_CFC_ (* Continuous Function Chart, elements in execution order *)
(* VÄRMEREGLERING *)
(* PUMPSTYRNING *)
(* BÖRVÄRDESKURVA *)
(* LARM/AVVIKELSELARM *)
#0 HUS1_VS20_SO(bManover: HUS2_AS01_SOMMARVINTER.bVINTER_TILL)
#1 HUS1_VS20_PV01(_bAuto: #0.bTILL)
#2 HUS1_VS20_PV01_M <= #1._bMANOVER
#3 HUS1_VS20_PV01_LD <= #1._bDRIFTFEL
#4 HUS1_VS20_PV01_LM <= #1._bLHAND
#5 SUB(HUS1_VS20_GT11_BB, HUS1_VS20_GT11_BB1)
#6 HUS1_VS20_GT11_PID(_bEnable: #0.bTILL, _rBV: #5, _rMV: HUS1_VS20_GT11_MV)
#7 HUS1_VS20_SV21_R <= #6._rY1
#8 HUS1_VS20_GT11_KURVA(_rGT3N: HUS2_AS01_GT31_MV)
#9 HUS1_VS20_GT11_BB <= #8._rBB
#10 HUS1_VS20_EFFEKTBEGR(_rGT3N: HUS2_AS01_GT31_MV, _rMQ41_SV: HUS2_VP1.SV_MQ41)
#11 HUS1_VS20_GT11_BB1 <= #10._rBB
#12 HUS1_VS20_GT11_larm()
_END_CFC_
(* the same logic as Structured Text *)
(* VÄRMEREGLERING *)
(* PUMPSTYRNING *)
(* BÖRVÄRDESKURVA *)
(* LARM/AVVIKELSELARM *)
HUS1_VS20_SO(bManover := HUS2_AS01_SOMMARVINTER.bVINTER_TILL);
HUS1_VS20_PV01(_bAuto := HUS1_VS20_SO.bTILL);
HUS1_VS20_PV01_M := HUS1_VS20_PV01._bMANOVER;
HUS1_VS20_PV01_LD := HUS1_VS20_PV01._bDRIFTFEL;
HUS1_VS20_PV01_LM := HUS1_VS20_PV01._bLHAND;
HUS1_VS20_GT11_PID(_bEnable := HUS1_VS20_SO.bTILL, _rBV := HUS1_VS20_GT11_BB - HUS1_VS20_GT11_BB1, _rMV := HUS1_VS20_GT11_MV);
HUS1_VS20_SV21_R := HUS1_VS20_GT11_PID._rY1;
HUS1_VS20_GT11_KURVA(_rGT3N := HUS2_AS01_GT31_MV);
HUS1_VS20_GT11_BB := HUS1_VS20_GT11_KURVA._rBB;
HUS1_VS20_EFFEKTBEGR(_rGT3N := HUS2_AS01_GT31_MV, _rMQ41_SV := HUS2_VP1.SV_MQ41);
HUS1_VS20_GT11_BB1 := HUS1_VS20_EFFEKTBEGR._rBB;
HUS1_VS20_GT11_larm();
END_PROGRAM

(* POU SYSTEM/VS20/HUS1_VS20_SO, CFC *)
PROGRAM HUS1_VS20_SO
VAR_INPUT

	bManover: BOOL;
END_VAR

VAR
	SERVICEOMKOPPLARE: fbManualOverride;

	UPPSTARTSSEKVENSIERING: BOOL;
END_VAR

VAR_OUTPUT
	bTILL:BOOL;

END_VAR
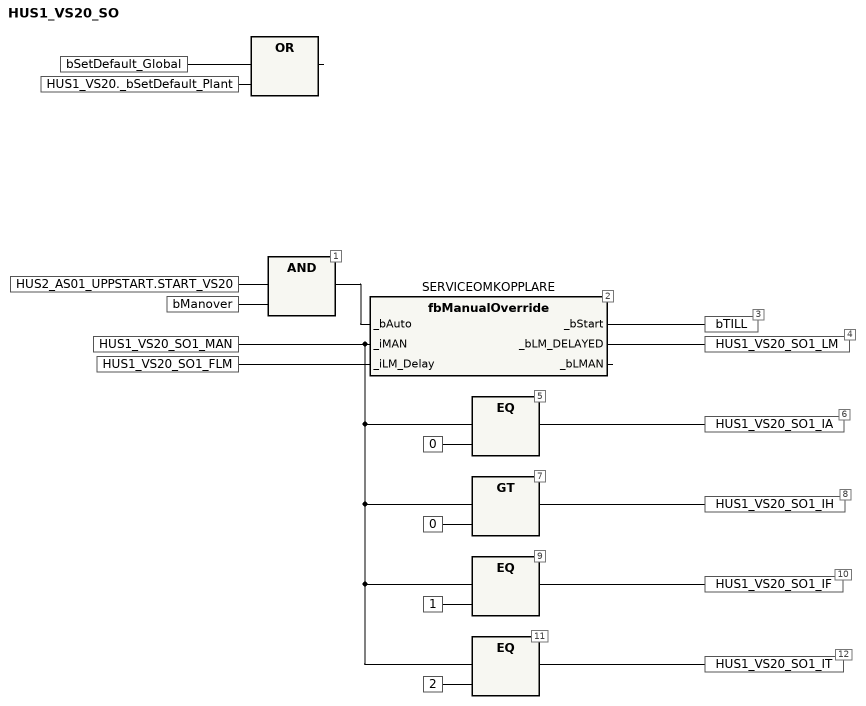
_CFC_ (* Continuous Function Chart, elements in execution order *)
#0 OR(bSetDefault_Global, HUS1_VS20._bSetDefault_Plant)
#1 AND(HUS2_AS01_UPPSTART.START_VS20, bManover)
#2 SERVICEOMKOPPLARE:fbManualOverride(_bAuto: #1, _iMAN: HUS1_VS20_SO1_MAN, _iLM_Delay: HUS1_VS20_SO1_FLM)
#3 bTILL <= #2._bStart
#4 HUS1_VS20_SO1_LM <= #2._bLM_DELAYED
#5 EQ(HUS1_VS20_SO1_MAN, 0)
#6 HUS1_VS20_SO1_IA <= #5
#7 GT(HUS1_VS20_SO1_MAN, 0)
#8 HUS1_VS20_SO1_IH <= #7
#9 EQ(HUS1_VS20_SO1_MAN, 1)
#10 HUS1_VS20_SO1_IF <= #9
#11 EQ(HUS1_VS20_SO1_MAN, 2)
#12 HUS1_VS20_SO1_IT <= #11
_END_CFC_
(* the same logic as Structured Text *)
(* result unused: bSetDefault_Global OR HUS1_VS20._bSetDefault_Plant *)
SERVICEOMKOPPLARE(_bAuto := HUS2_AS01_UPPSTART.START_VS20 AND bManover, _iMAN := HUS1_VS20_SO1_MAN, _iLM_Delay := HUS1_VS20_SO1_FLM);
bTILL := SERVICEOMKOPPLARE._bStart;
HUS1_VS20_SO1_LM := SERVICEOMKOPPLARE._bLM_DELAYED;
HUS1_VS20_SO1_IA := HUS1_VS20_SO1_MAN = 0;
HUS1_VS20_SO1_IH := HUS1_VS20_SO1_MAN > 0;
HUS1_VS20_SO1_IF := HUS1_VS20_SO1_MAN = 1;
HUS1_VS20_SO1_IT := HUS1_VS20_SO1_MAN = 2;
END_PROGRAM

(* POU SYSTEM/VS20/Pumpstyrning/HUS1_VS20_PV01, CFC *)
PROGRAM HUS1_VS20_PV01

VAR

	Default: BOOL;
	Motor: FB_HVACMotor1Speed;


	fbReset1: fbBool_Reset;
	AlarmDelay: fbDelayedAlarmSeconds;

	MANHAND: fbManualOverride;
END_VAR
VAR


(********************MOTOR********************)
(*INPUT*)
	eCtrlModeActuator			:E_HVACActuatorMode;
	tStartDelay						:TIME;
	tStopDelay						:TIME;
	tDelayFeedbContactor			:TIME:=T#30s;
	tFeedbProcessTimer				:TIME:=T#30s;
	tDelayFeedbProcess				:TIME:=T#30s;
(*OUTPUT*)
	byState							:BYTE ;
	bStateAuto							:BOOL;
	bStateRepairSwitch				:BOOL;
	bStateManSwitch				:BOOL;
	eStateModeActuator				:E_HVACActuatorMode;
	byError							:BYTE ;
	bErrorMotorprotec				:BOOL;
	bErrorFeedbContactor			:BOOL;
	bErrorFeedbProcess			:BOOL;
	bInvalidParameter				:BOOL;

END_VAR

VAR_INPUT
	_bAuto							:BOOL;(* enable function block *)
END_VAR

VAR_OUTPUT
	_bMANOVER						:BOOL;
	_bDRIFTFEL						:BOOL;
	_bLHAND							:BOOL;
END_VAR
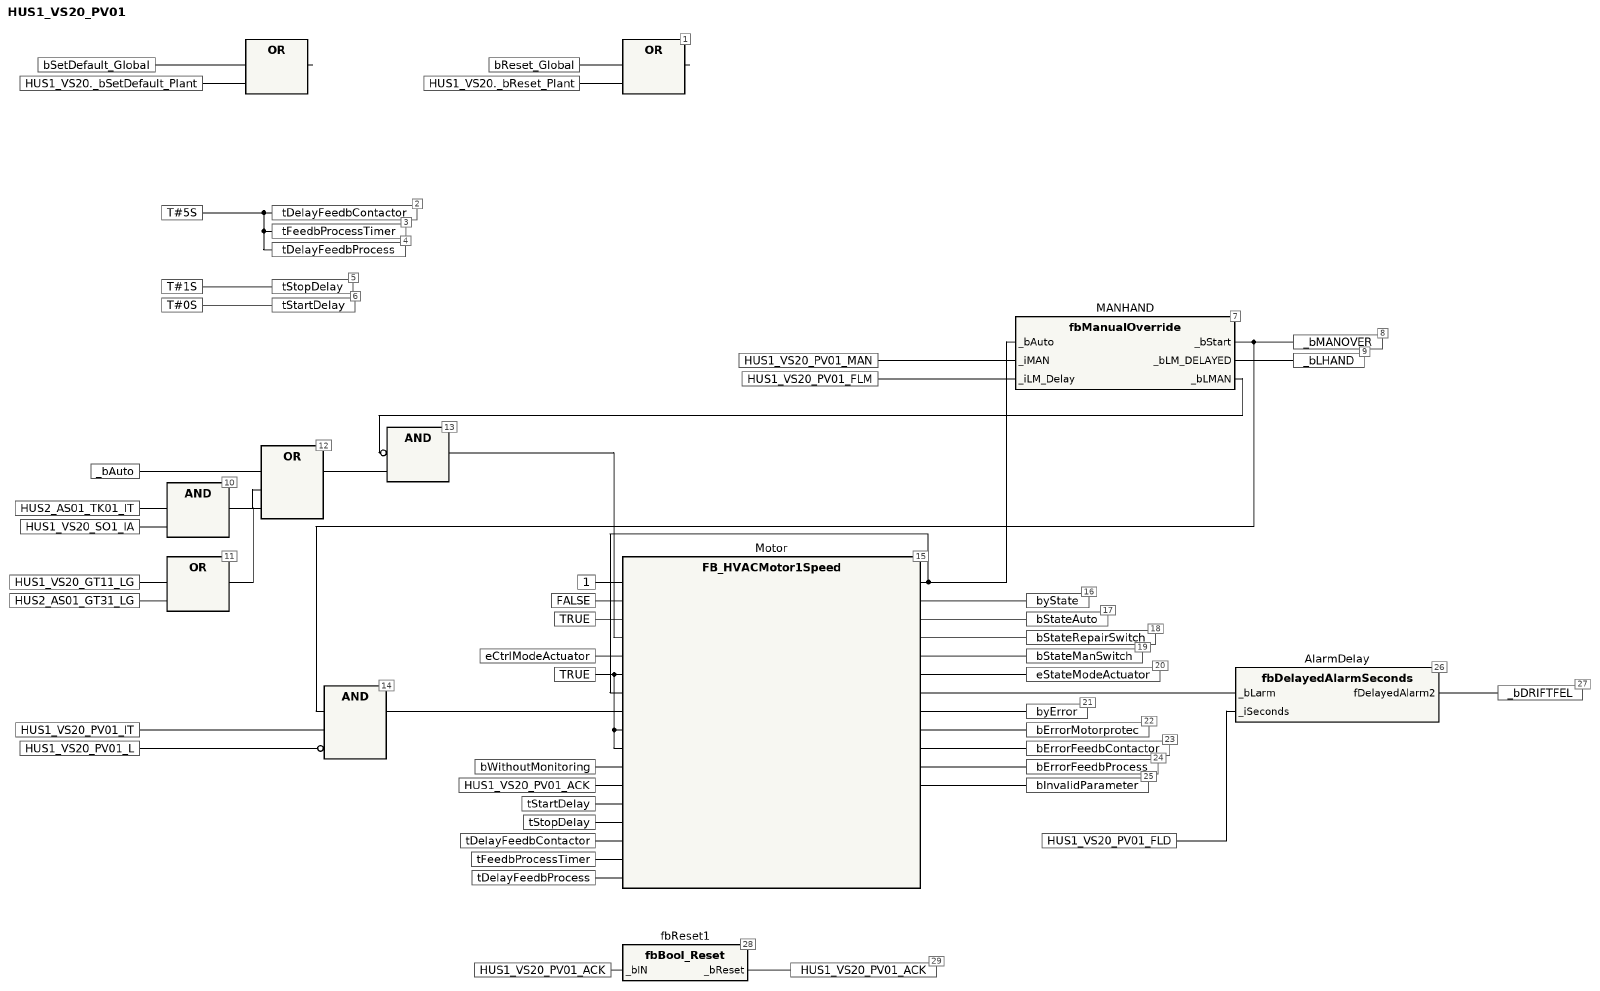
_CFC_ (* Continuous Function Chart, elements in execution order *)
#0 OR(bSetDefault_Global, HUS1_VS20._bSetDefault_Plant)
#1 OR(bReset_Global, HUS1_VS20._bReset_Plant)
#2 tDelayFeedbContactor <= T#5S
#3 tFeedbProcessTimer <= T#5S
#4 tDelayFeedbProcess <= T#5S
#5 tStopDelay <= T#1S
#6 tStartDelay <= T#0S
#7 MANHAND:fbManualOverride(_bAuto: #15.out 1, _iMAN: HUS1_VS20_PV01_MAN, _iLM_Delay: HUS1_VS20_PV01_FLM)
#8 _bMANOVER <= #7._bStart
#9 _bLHAND <= #7._bLM_DELAYED
#10 AND(HUS2_AS01_TK01_IT, HUS1_VS20_SO1_IA)
#11 OR(HUS1_VS20_GT11_LG, HUS2_AS01_GT31_LG)
#12 OR(_bAuto, #10, #11)
#13 AND(NOT #7._bLMAN, #12)
#14 AND(#7._bStart, HUS1_VS20_PV01_IT, NOT HUS1_VS20_PV01_L)
#15 Motor:FB_HVACMotor1Speed(1, FALSE, TRUE, #13, eCtrlModeActuator, TRUE, #15.out 1, #14, TRUE, TRUE, bWithoutMonitoring, HUS1_VS20_PV01_ACK, tStartDelay, tStopDelay, tDelayFeedbContactor, tFeedbProcessTimer, tDelayFeedbProcess)
#16 byState <= #15.out 2
#17 bStateAuto <= #15.out 3
#18 bStateRepairSwitch <= #15.out 4
#19 bStateManSwitch <= #15.out 5
#20 eStateModeActuator <= #15.out 6
#21 byError <= #15.out 8
#22 bErrorMotorprotec <= #15.out 9
#23 bErrorFeedbContactor <= #15.out 10
#24 bErrorFeedbProcess <= #15.out 11
#25 bInvalidParameter <= #15.out 12
#26 AlarmDelay:fbDelayedAlarmSeconds(_bLarm: #15.out 7, _iSeconds: HUS1_VS20_PV01_FLD)
#27 _bDRIFTFEL <= #26.fDelayedAlarm2
#28 fbReset1:fbBool_Reset(_bIN: HUS1_VS20_PV01_ACK)
#29 HUS1_VS20_PV01_ACK <= #28._bReset
_END_CFC_
END_PROGRAM

(* POU SYSTEM/VS20/Tempreglering/HUS1_VS20_GT11_PID, FAI *)
PROGRAM HUS1_VS20_GT11_PID

VAR_INPUT
	_bEnable		:BOOL;
	_rBV			:REAL;
	_rMV			:REAL;
END_VAR

VAR_OUTPUT
	_rY1                         : REAL;
END_VAR


VAR
	_bSetDefaultPID:BOOL;
	_bReset_Local:BOOL;


	SVX: FB_HVACPIDCtrl;
	eDataSecurityType         : E_HVACDataSecurityType;
	rInitialValue            : REAL;
	bResetController          : BOOL;
	_eCtrlMode				:E_HVACCtrlMode;(*
									eHVACCtrlMode_Auto      := 0,
								   	eHVACCtrlMode_Manual   := 1 *)
	_rOverrideValue			:REAL;(* controller output rY in operating mode eCtrlMode =1 *)
	rXW                        : REAL;
	bMaxLimit                  : BOOL;
	bMinLimit                  : BOOL;
	bActive                    : BOOL;
	bARWactive                 : BOOL;
	eState                     : E_HVACState;
	bError                     : BOOL;
	eErrorCode                 : E_HVACErrorCodes;
	bInvalidParameter          : BOOL;

	bDirection              : BOOL;
	_rKP: REAL;
	_rCH: REAL;
	tTi                     : TIME;
	tTv                     : TIME;
	tTd                     : TIME;

	rYMin                   : REAL;
	rYMax                   : REAL;

	CI: fbBer_PID_inst;
	CS: fbBer_PID_inst;
	CD: fbBer_PID_inst;

	fbPersistent_CH: FB_HVACPersistent_Real;
	fbPersistent_CP: FB_HVACPersistent_Real;
	fbPersistent_CI: FB_HVACPersistent_Real;
	fbPersistent_CS: FB_HVACPersistent_Real;
	fbPersistent_CD: FB_HVACPersistent_Real;
	LM_DELAY: fbDelayedAlarmMinutes;
END_VAR
(* body not read: cfc97 *)
END_PROGRAM

(* POU SYSTEM/VS20/Börvärden & kurvor/HUS1_VS20_GT11_KURVA, FAI *)
PROGRAM HUS1_VS20_GT11_KURVA
VAR
(****************************************** heating curve **********************************************************************************************************************)

	_bSetDefaultHC			:BOOL;


	fbScale_n:			FB_HVACScale_nPoint;
	_bErrParam:			BOOL;								(*ParameterError*)
	stScaleParameter:	ST_HVACParameterScale_nPoint	;	(*Parameter struktur på antal brutpunkter*)


	fbTemp1:	FB_HVACPersistent_Real;
	fbTemp2:	FB_HVACPersistent_Real;
	fbTemp3:	FB_HVACPersistent_Real;
	fbTemp4:	FB_HVACPersistent_Real;
	fbTemp5:	FB_HVACPersistent_Real;

	fbOutsideTemp1:	FB_HVACPersistent_Real;
	fbOutsideTemp2:	FB_HVACPersistent_Real;
	fbOutsideTemp3:	FB_HVACPersistent_Real;
	fbOutsideTemp4:	FB_HVACPersistent_Real;
	fbOutsideTemp5:	FB_HVACPersistent_Real;
	BB_min: FB_HVACPersistent_Real;
	BB_max: FB_HVACPersistent_Real;

END_VAR

VAR_INPUT
	_rGT3N	:REAL; (*Utegivare*)

END_VAR

VAR_OUTPUT
	_rBB		:LREAL;
END_VAR
(* body not read: cfc97 *)
END_PROGRAM

(* POU SYSTEM/VS20/Börvärden & kurvor/HUS1_VS20_EFFEKTBEGR, FAI *)
PROGRAM HUS1_VS20_EFFEKTBEGR
VAR
(****************************************** heating curve **********************************************************************************************************************)

	_bSetDefaultHC			:BOOL;


	fbScale_n:			FB_HVACScale_nPoint;
	_bErrParam:			BOOL;								(*ParameterError*)
	stScaleParameter:	ST_HVACParameterScale_nPoint	;	(*Parameter struktur på antal brutpunkter*)


	fbTemp1:	FB_HVACPersistent_Real;
	fbTemp2:	FB_HVACPersistent_Real;
	fbTemp3:	FB_HVACPersistent_Real;
	fbTemp4:	FB_HVACPersistent_Real;
	fbTemp5:	FB_HVACPersistent_Real;

	fbOutsideTemp1:	FB_HVACPersistent_Real;
	fbOutsideTemp2:	FB_HVACPersistent_Real;
	fbOutsideTemp3:	FB_HVACPersistent_Real;
	fbOutsideTemp4:	FB_HVACPersistent_Real;
	fbOutsideTemp5:	FB_HVACPersistent_Real;
	BB_min: FB_HVACPersistent_Real;
	BB_max: FB_HVACPersistent_Real;

	CalcForskjutning: fbConversionScale;
	MIN_LIMIT: REAL;
END_VAR

VAR_INPUT
	_rGT3N	:REAL; (*Utegivare*)
	_rMQ41_SV	:REAL;

END_VAR

VAR_OUTPUT
	_rBB		:LREAL;
END_VAR
(* body not read: cfc97 *)
END_PROGRAM

(* POU SYSTEM/VS20/Larm/HUS1_VS20_GT11_LARM, FAI *)
PROGRAM HUS1_VS20_GT11_LARM

VAR_OUTPUT
	_bLSumma					: BOOL;	(*Summalarm*)

END_VAR
VAR

	_bSetDefault: 				BOOL;		(*Se default values*)
	fbLarm: fbAvvikelselarm;


	fbHigh: FB_HVACPersistent_Real;
	fbAlarmDelayLH: FB_HVACPersistent_Int;
	fbLow: FB_HVACPersistent_Real;
	fbAlarmDelayLL: FB_HVACPersistent_Int;


END_VAR
(* body not read: cfc97 *)
END_PROGRAM

(* POU SYSTEM/VS30/HUS2_VS30, CFC *)
PROGRAM HUS2_VS30
VAR
	_bSetDefault_Plant		:BOOL;
	_bReset_Plant				:BOOL;

END_VAR
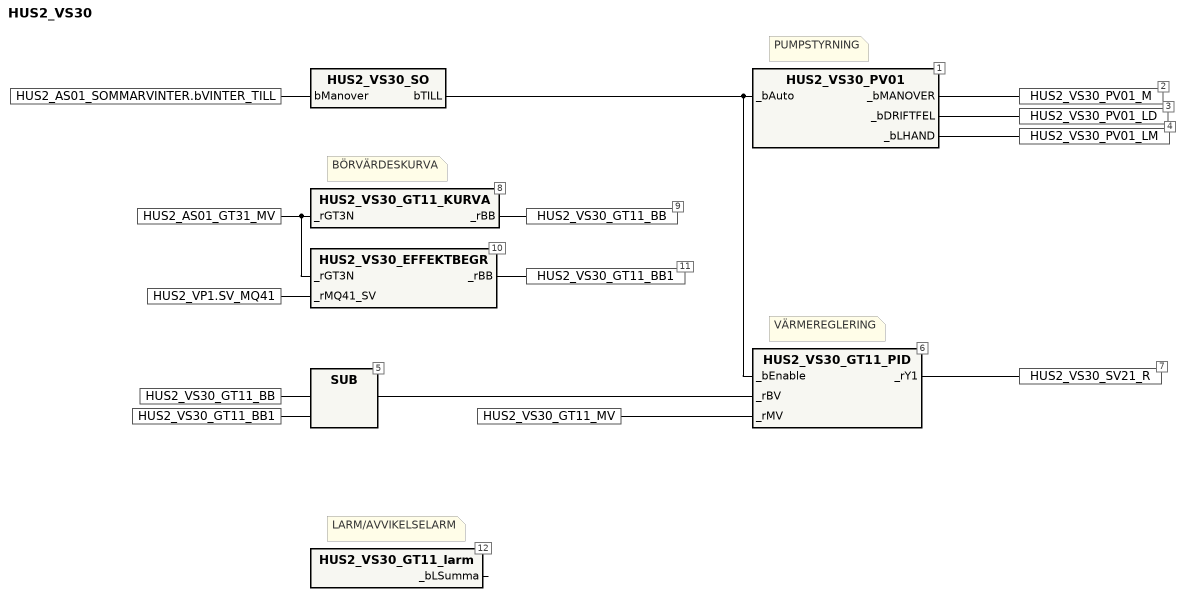
_CFC_ (* Continuous Function Chart, elements in execution order *)
(* LARM/AVVIKELSELARM *)
(* BÖRVÄRDESKURVA *)
(* PUMPSTYRNING *)
(* VÄRMEREGLERING *)
#0 HUS2_VS30_SO(bManover: HUS2_AS01_SOMMARVINTER.bVINTER_TILL)
#1 HUS2_VS30_PV01(_bAuto: #0.bTILL)
#2 HUS2_VS30_PV01_M <= #1._bMANOVER
#3 HUS2_VS30_PV01_LD <= #1._bDRIFTFEL
#4 HUS2_VS30_PV01_LM <= #1._bLHAND
#5 SUB(HUS2_VS30_GT11_BB, HUS2_VS30_GT11_BB1)
#6 HUS2_VS30_GT11_PID(_bEnable: #0.bTILL, _rBV: #5, _rMV: HUS2_VS30_GT11_MV)
#7 HUS2_VS30_SV21_R <= #6._rY1
#8 HUS2_VS30_GT11_KURVA(_rGT3N: HUS2_AS01_GT31_MV)
#9 HUS2_VS30_GT11_BB <= #8._rBB
#10 HUS2_VS30_EFFEKTBEGR(_rGT3N: HUS2_AS01_GT31_MV, _rMQ41_SV: HUS2_VP1.SV_MQ41)
#11 HUS2_VS30_GT11_BB1 <= #10._rBB
#12 HUS2_VS30_GT11_larm()
_END_CFC_
(* the same logic as Structured Text *)
(* LARM/AVVIKELSELARM *)
(* BÖRVÄRDESKURVA *)
(* PUMPSTYRNING *)
(* VÄRMEREGLERING *)
HUS2_VS30_SO(bManover := HUS2_AS01_SOMMARVINTER.bVINTER_TILL);
HUS2_VS30_PV01(_bAuto := HUS2_VS30_SO.bTILL);
HUS2_VS30_PV01_M := HUS2_VS30_PV01._bMANOVER;
HUS2_VS30_PV01_LD := HUS2_VS30_PV01._bDRIFTFEL;
HUS2_VS30_PV01_LM := HUS2_VS30_PV01._bLHAND;
HUS2_VS30_GT11_PID(_bEnable := HUS2_VS30_SO.bTILL, _rBV := HUS2_VS30_GT11_BB - HUS2_VS30_GT11_BB1, _rMV := HUS2_VS30_GT11_MV);
HUS2_VS30_SV21_R := HUS2_VS30_GT11_PID._rY1;
HUS2_VS30_GT11_KURVA(_rGT3N := HUS2_AS01_GT31_MV);
HUS2_VS30_GT11_BB := HUS2_VS30_GT11_KURVA._rBB;
HUS2_VS30_EFFEKTBEGR(_rGT3N := HUS2_AS01_GT31_MV, _rMQ41_SV := HUS2_VP1.SV_MQ41);
HUS2_VS30_GT11_BB1 := HUS2_VS30_EFFEKTBEGR._rBB;
HUS2_VS30_GT11_larm();
END_PROGRAM

(* POU SYSTEM/VS30/HUS2_VS30_SO, CFC *)
PROGRAM HUS2_VS30_SO
VAR_INPUT

	bManover: BOOL;
END_VAR

VAR
	SERVICEOMKOPPLARE: fbManualOverride;

	UPPSTARTSSEKVENSIERING: BOOL;
END_VAR

VAR_OUTPUT
	bTILL:BOOL;

END_VAR
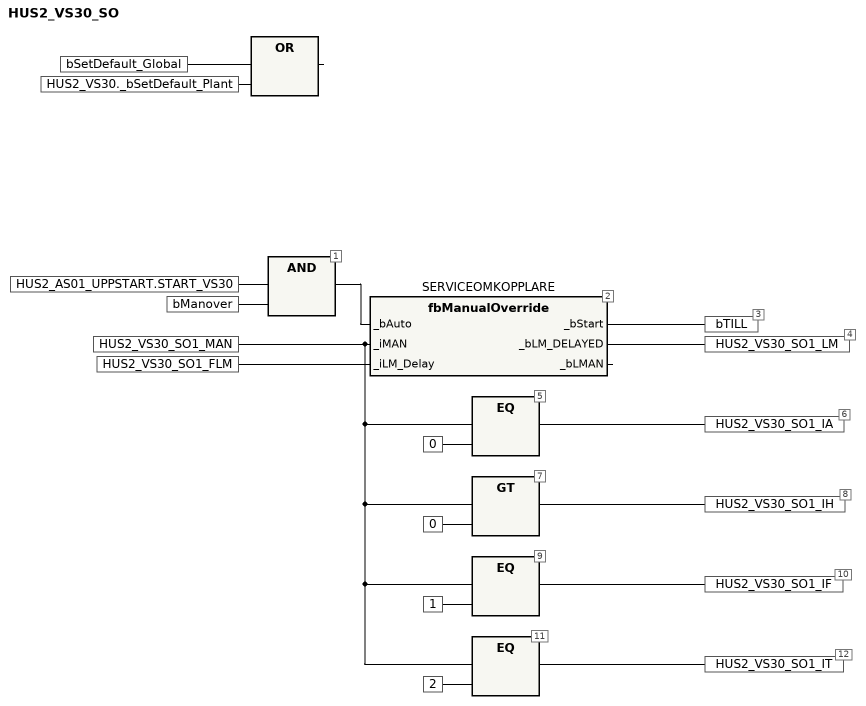
_CFC_ (* Continuous Function Chart, elements in execution order *)
#0 OR(bSetDefault_Global, HUS2_VS30._bSetDefault_Plant)
#1 AND(HUS2_AS01_UPPSTART.START_VS30, bManover)
#2 SERVICEOMKOPPLARE:fbManualOverride(_bAuto: #1, _iMAN: HUS2_VS30_SO1_MAN, _iLM_Delay: HUS2_VS30_SO1_FLM)
#3 bTILL <= #2._bStart
#4 HUS2_VS30_SO1_LM <= #2._bLM_DELAYED
#5 EQ(HUS2_VS30_SO1_MAN, 0)
#6 HUS2_VS30_SO1_IA <= #5
#7 GT(HUS2_VS30_SO1_MAN, 0)
#8 HUS2_VS30_SO1_IH <= #7
#9 EQ(HUS2_VS30_SO1_MAN, 1)
#10 HUS2_VS30_SO1_IF <= #9
#11 EQ(HUS2_VS30_SO1_MAN, 2)
#12 HUS2_VS30_SO1_IT <= #11
_END_CFC_
(* the same logic as Structured Text *)
(* result unused: bSetDefault_Global OR HUS2_VS30._bSetDefault_Plant *)
SERVICEOMKOPPLARE(_bAuto := HUS2_AS01_UPPSTART.START_VS30 AND bManover, _iMAN := HUS2_VS30_SO1_MAN, _iLM_Delay := HUS2_VS30_SO1_FLM);
bTILL := SERVICEOMKOPPLARE._bStart;
HUS2_VS30_SO1_LM := SERVICEOMKOPPLARE._bLM_DELAYED;
HUS2_VS30_SO1_IA := HUS2_VS30_SO1_MAN = 0;
HUS2_VS30_SO1_IH := HUS2_VS30_SO1_MAN > 0;
HUS2_VS30_SO1_IF := HUS2_VS30_SO1_MAN = 1;
HUS2_VS30_SO1_IT := HUS2_VS30_SO1_MAN = 2;
END_PROGRAM

(* POU SYSTEM/VS30/Pumpstyrning/HUS2_VS30_PV01, CFC *)
PROGRAM HUS2_VS30_PV01

VAR

	Default: BOOL;
	Motor: FB_HVACMotor1Speed;


	fbReset1: fbBool_Reset;
	AlarmDelay: fbDelayedAlarmSeconds;

	MANHAND: fbManualOverride;
END_VAR
VAR


(********************MOTOR********************)
(*INPUT*)
	eCtrlModeActuator			:E_HVACActuatorMode;
	tStartDelay						:TIME;
	tStopDelay						:TIME;
	tDelayFeedbContactor			:TIME:=T#30s;
	tFeedbProcessTimer				:TIME:=T#30s;
	tDelayFeedbProcess				:TIME:=T#30s;
(*OUTPUT*)
	byState							:BYTE ;
	bStateAuto							:BOOL;
	bStateRepairSwitch				:BOOL;
	bStateManSwitch				:BOOL;
	eStateModeActuator				:E_HVACActuatorMode;
	byError							:BYTE ;
	bErrorMotorprotec				:BOOL;
	bErrorFeedbContactor			:BOOL;
	bErrorFeedbProcess			:BOOL;
	bInvalidParameter				:BOOL;

END_VAR

VAR_INPUT
	_bAuto							:BOOL;(* enable function block *)
END_VAR

VAR_OUTPUT
	_bMANOVER						:BOOL;
	_bDRIFTFEL						:BOOL;
	_bLHAND							:BOOL;
END_VAR
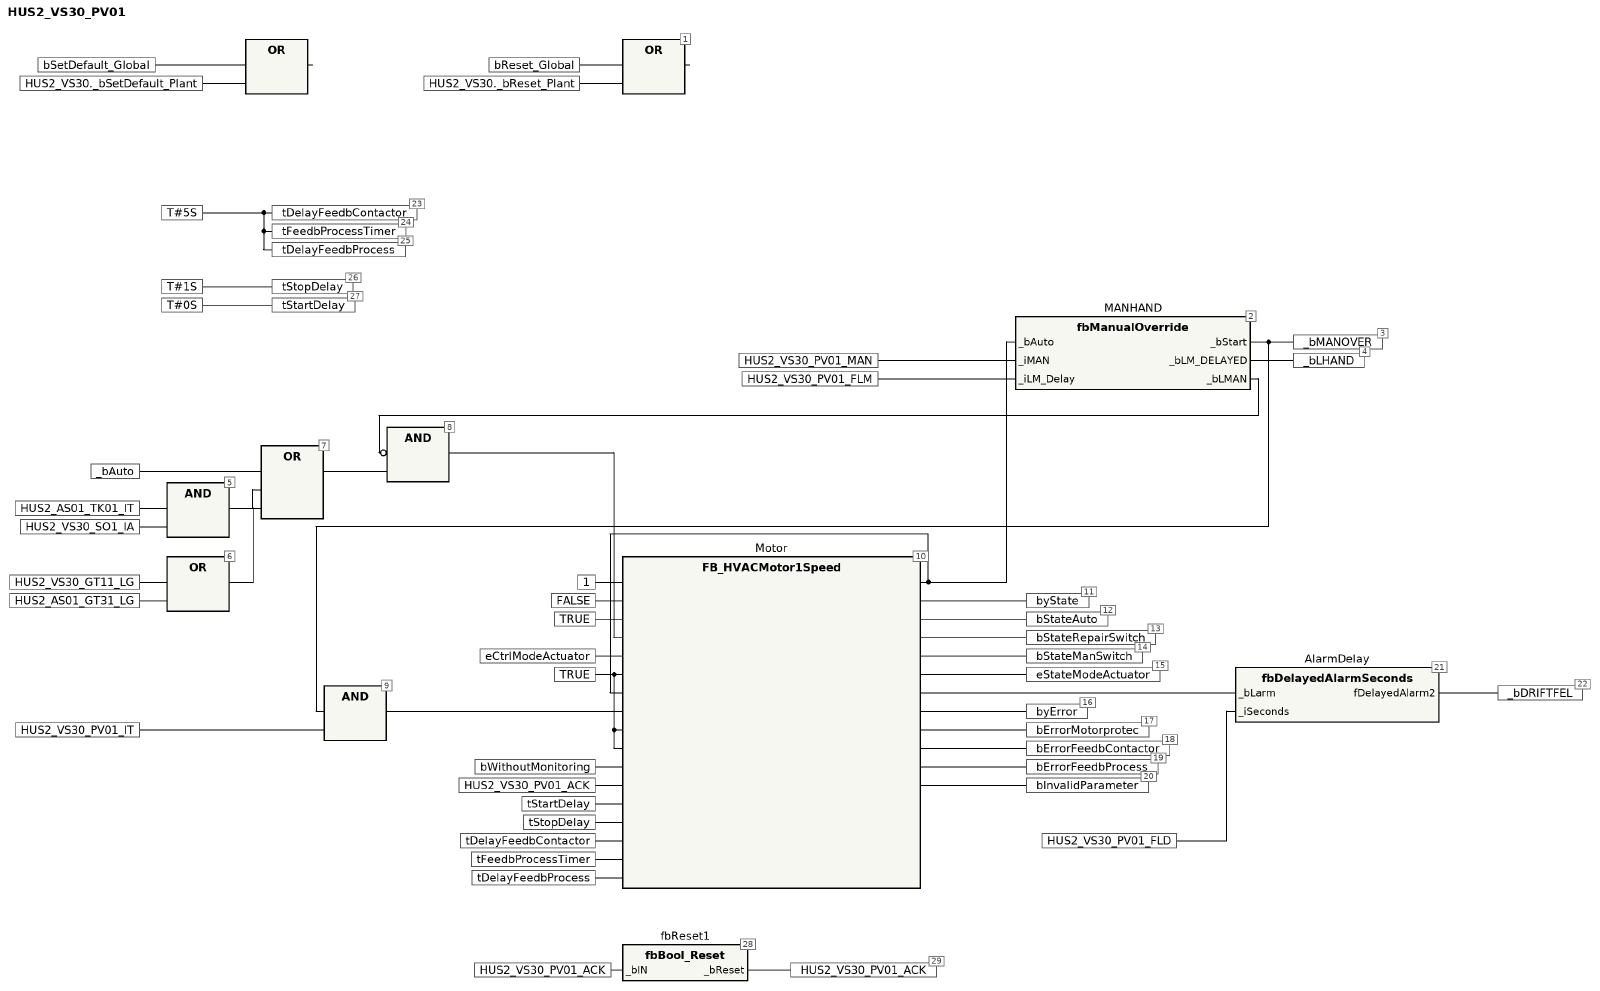
_CFC_ (* Continuous Function Chart, elements in execution order *)
#0 OR(bSetDefault_Global, HUS2_VS30._bSetDefault_Plant)
#1 OR(bReset_Global, HUS2_VS30._bReset_Plant)
#2 MANHAND:fbManualOverride(_bAuto: #10.out 1, _iMAN: HUS2_VS30_PV01_MAN, _iLM_Delay: HUS2_VS30_PV01_FLM)
#3 _bMANOVER <= #2._bStart
#4 _bLHAND <= #2._bLM_DELAYED
#5 AND(HUS2_AS01_TK01_IT, HUS2_VS30_SO1_IA)
#6 OR(HUS2_VS30_GT11_LG, HUS2_AS01_GT31_LG)
#7 OR(_bAuto, #5, #6)
#8 AND(NOT #2._bLMAN, #7)
#9 AND(#2._bStart, HUS2_VS30_PV01_IT)
#10 Motor:FB_HVACMotor1Speed(1, FALSE, TRUE, #8, eCtrlModeActuator, TRUE, #10.out 1, #9, TRUE, TRUE, bWithoutMonitoring, HUS2_VS30_PV01_ACK, tStartDelay, tStopDelay, tDelayFeedbContactor, tFeedbProcessTimer, tDelayFeedbProcess)
#11 byState <= #10.out 2
#12 bStateAuto <= #10.out 3
#13 bStateRepairSwitch <= #10.out 4
#14 bStateManSwitch <= #10.out 5
#15 eStateModeActuator <= #10.out 6
#16 byError <= #10.out 8
#17 bErrorMotorprotec <= #10.out 9
#18 bErrorFeedbContactor <= #10.out 10
#19 bErrorFeedbProcess <= #10.out 11
#20 bInvalidParameter <= #10.out 12
#21 AlarmDelay:fbDelayedAlarmSeconds(_bLarm: #10.out 7, _iSeconds: HUS2_VS30_PV01_FLD)
#22 _bDRIFTFEL <= #21.fDelayedAlarm2
#23 tDelayFeedbContactor <= T#5S
#24 tFeedbProcessTimer <= T#5S
#25 tDelayFeedbProcess <= T#5S
#26 tStopDelay <= T#1S
#27 tStartDelay <= T#0S
#28 fbReset1:fbBool_Reset(_bIN: HUS2_VS30_PV01_ACK)
#29 HUS2_VS30_PV01_ACK <= #28._bReset
_END_CFC_
END_PROGRAM

(* POU SYSTEM/VS30/Tempreglering/HUS2_VS30_GT11_PID, FAI *)
PROGRAM HUS2_VS30_GT11_PID

VAR_INPUT
	_bEnable		:BOOL;
	_rBV			:REAL;
	_rMV			:REAL;
END_VAR

VAR_OUTPUT
	_rY1                         : REAL;
END_VAR


VAR
	_bSetDefaultPID:BOOL;
	_bReset_Local:BOOL;


	SVX: FB_HVACPIDCtrl;
	eDataSecurityType         : E_HVACDataSecurityType;
	rInitialValue            : REAL;
	bResetController          : BOOL;
	_eCtrlMode				:E_HVACCtrlMode;(*
									eHVACCtrlMode_Auto      := 0,
								   	eHVACCtrlMode_Manual   := 1 *)
	_rOverrideValue			:REAL;(* controller output rY in operating mode eCtrlMode =1 *)
	rXW                        : REAL;
	bMaxLimit                  : BOOL;
	bMinLimit                  : BOOL;
	bActive                    : BOOL;
	bARWactive                 : BOOL;
	eState                     : E_HVACState;
	bError                     : BOOL;
	eErrorCode                 : E_HVACErrorCodes;
	bInvalidParameter          : BOOL;

	bDirection              : BOOL;
	_rKP: REAL;
	_rCH: REAL;
	tTi                     : TIME;
	tTv                     : TIME;
	tTd                     : TIME;

	rYMin                   : REAL;
	rYMax                   : REAL;

	CI: fbBer_PID_inst;
	CS: fbBer_PID_inst;
	CD: fbBer_PID_inst;

	fbPersistent_CH: FB_HVACPersistent_Real;
	fbPersistent_CP: FB_HVACPersistent_Real;
	fbPersistent_CI: FB_HVACPersistent_Real;
	fbPersistent_CS: FB_HVACPersistent_Real;
	fbPersistent_CD: FB_HVACPersistent_Real;
	LM_DELAY: fbDelayedAlarmMinutes;
END_VAR
(* body not read: cfc97 *)
END_PROGRAM

(* POU SYSTEM/VS30/Börvärden & kurvor/HUS2_VS30_GT11_KURVA, FAI *)
PROGRAM HUS2_VS30_GT11_KURVA
VAR
(****************************************** heating curve **********************************************************************************************************************)

	_bSetDefaultHC			:BOOL;


	fbScale_n:			FB_HVACScale_nPoint;
	_bErrParam:			BOOL;								(*ParameterError*)
	stScaleParameter:	ST_HVACParameterScale_nPoint	;	(*Parameter struktur på antal brutpunkter*)


	fbTemp1:	FB_HVACPersistent_Real;
	fbTemp2:	FB_HVACPersistent_Real;
	fbTemp3:	FB_HVACPersistent_Real;
	fbTemp4:	FB_HVACPersistent_Real;
	fbTemp5:	FB_HVACPersistent_Real;

	fbOutsideTemp1:	FB_HVACPersistent_Real;
	fbOutsideTemp2:	FB_HVACPersistent_Real;
	fbOutsideTemp3:	FB_HVACPersistent_Real;
	fbOutsideTemp4:	FB_HVACPersistent_Real;
	fbOutsideTemp5:	FB_HVACPersistent_Real;
	BB_min: FB_HVACPersistent_Real;
	BB_max: FB_HVACPersistent_Real;

END_VAR

VAR_INPUT
	_rGT3N	:REAL; (*Utegivare*)

END_VAR

VAR_OUTPUT
	_rBB		:LREAL;
END_VAR
(* body not read: cfc97 *)
END_PROGRAM

(* POU SYSTEM/VS30/Börvärden & kurvor/HUS2_VS30_EFFEKTBEGR, FAI *)
PROGRAM HUS2_VS30_EFFEKTBEGR
VAR
(****************************************** heating curve **********************************************************************************************************************)

	_bSetDefaultHC			:BOOL;


	fbScale_n:			FB_HVACScale_nPoint;
	_bErrParam:			BOOL;								(*ParameterError*)
	stScaleParameter:	ST_HVACParameterScale_nPoint	;	(*Parameter struktur på antal brutpunkter*)


	fbTemp1:	FB_HVACPersistent_Real;
	fbTemp2:	FB_HVACPersistent_Real;
	fbTemp3:	FB_HVACPersistent_Real;
	fbTemp4:	FB_HVACPersistent_Real;
	fbTemp5:	FB_HVACPersistent_Real;

	fbOutsideTemp1:	FB_HVACPersistent_Real;
	fbOutsideTemp2:	FB_HVACPersistent_Real;
	fbOutsideTemp3:	FB_HVACPersistent_Real;
	fbOutsideTemp4:	FB_HVACPersistent_Real;
	fbOutsideTemp5:	FB_HVACPersistent_Real;
	BB_min: FB_HVACPersistent_Real;
	BB_max: FB_HVACPersistent_Real;

	CalcForskjutning: fbConversionScale;
	MIN_LIMIT: REAL;
END_VAR

VAR_INPUT
	_rGT3N	:REAL; (*Utegivare*)
	_rMQ41_SV	:REAL;

END_VAR

VAR_OUTPUT
	_rBB		:LREAL;
END_VAR
(* body not read: cfc97 *)
END_PROGRAM

(* POU SYSTEM/VS30/Larm/HUS2_VS30_GT11_LARM, FAI *)
PROGRAM HUS2_VS30_GT11_LARM

VAR_OUTPUT
	_bLSumma					: BOOL;	(*Summalarm*)

END_VAR
VAR

	_bSetDefault: 				BOOL;		(*Se default values*)
	fbLarm: fbAvvikelselarm;


	fbHigh: FB_HVACPersistent_Real;
	fbAlarmDelayLH: FB_HVACPersistent_Int;
	fbLow: FB_HVACPersistent_Real;
	fbAlarmDelayLL: FB_HVACPersistent_Int;


END_VAR
(* body not read: cfc97 *)
END_PROGRAM

(* POU SYSTEM/VS40/HUS3_VS40, CFC *)
PROGRAM HUS3_VS40
VAR
	_bSetDefault_Plant		:BOOL;
	_bReset_Plant				:BOOL;

END_VAR
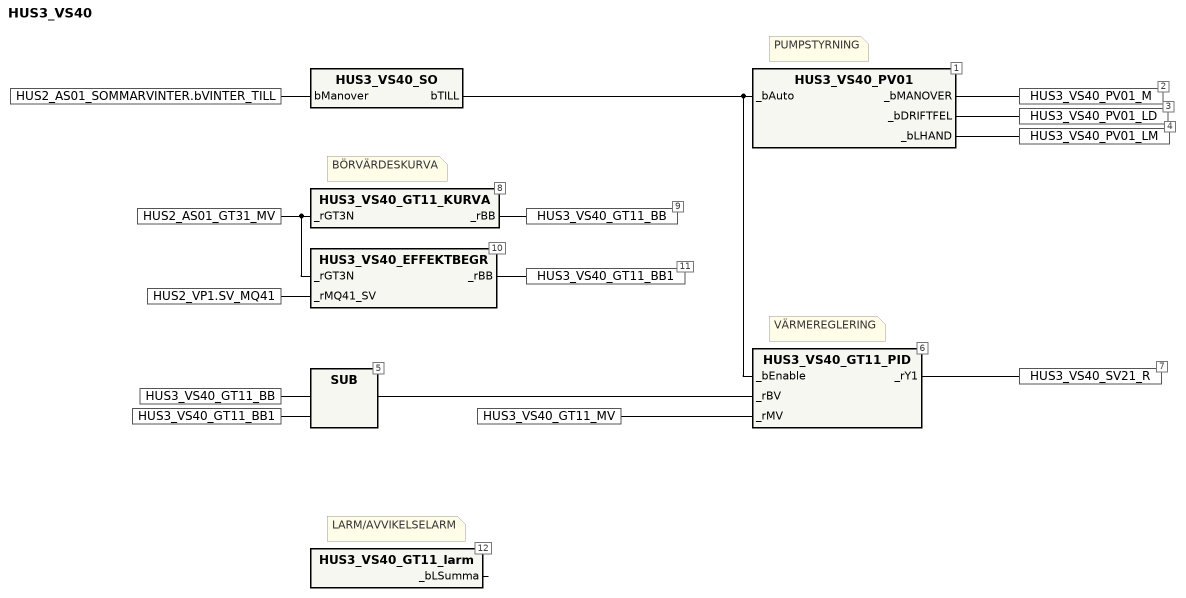
_CFC_ (* Continuous Function Chart, elements in execution order *)
(* VÄRMEREGLERING *)
(* PUMPSTYRNING *)
(* BÖRVÄRDESKURVA *)
(* LARM/AVVIKELSELARM *)
#0 HUS3_VS40_SO(bManover: HUS2_AS01_SOMMARVINTER.bVINTER_TILL)
#1 HUS3_VS40_PV01(_bAuto: #0.bTILL)
#2 HUS3_VS40_PV01_M <= #1._bMANOVER
#3 HUS3_VS40_PV01_LD <= #1._bDRIFTFEL
#4 HUS3_VS40_PV01_LM <= #1._bLHAND
#5 SUB(HUS3_VS40_GT11_BB, HUS3_VS40_GT11_BB1)
#6 HUS3_VS40_GT11_PID(_bEnable: #0.bTILL, _rBV: #5, _rMV: HUS3_VS40_GT11_MV)
#7 HUS3_VS40_SV21_R <= #6._rY1
#8 HUS3_VS40_GT11_KURVA(_rGT3N: HUS2_AS01_GT31_MV)
#9 HUS3_VS40_GT11_BB <= #8._rBB
#10 HUS3_VS40_EFFEKTBEGR(_rGT3N: HUS2_AS01_GT31_MV, _rMQ41_SV: HUS2_VP1.SV_MQ41)
#11 HUS3_VS40_GT11_BB1 <= #10._rBB
#12 HUS3_VS40_GT11_larm()
_END_CFC_
(* the same logic as Structured Text *)
(* VÄRMEREGLERING *)
(* PUMPSTYRNING *)
(* BÖRVÄRDESKURVA *)
(* LARM/AVVIKELSELARM *)
HUS3_VS40_SO(bManover := HUS2_AS01_SOMMARVINTER.bVINTER_TILL);
HUS3_VS40_PV01(_bAuto := HUS3_VS40_SO.bTILL);
HUS3_VS40_PV01_M := HUS3_VS40_PV01._bMANOVER;
HUS3_VS40_PV01_LD := HUS3_VS40_PV01._bDRIFTFEL;
HUS3_VS40_PV01_LM := HUS3_VS40_PV01._bLHAND;
HUS3_VS40_GT11_PID(_bEnable := HUS3_VS40_SO.bTILL, _rBV := HUS3_VS40_GT11_BB - HUS3_VS40_GT11_BB1, _rMV := HUS3_VS40_GT11_MV);
HUS3_VS40_SV21_R := HUS3_VS40_GT11_PID._rY1;
HUS3_VS40_GT11_KURVA(_rGT3N := HUS2_AS01_GT31_MV);
HUS3_VS40_GT11_BB := HUS3_VS40_GT11_KURVA._rBB;
HUS3_VS40_EFFEKTBEGR(_rGT3N := HUS2_AS01_GT31_MV, _rMQ41_SV := HUS2_VP1.SV_MQ41);
HUS3_VS40_GT11_BB1 := HUS3_VS40_EFFEKTBEGR._rBB;
HUS3_VS40_GT11_larm();
END_PROGRAM

(* POU SYSTEM/VS40/HUS3_VS40_SO, CFC *)
PROGRAM HUS3_VS40_SO
VAR_INPUT

	bManover: BOOL;
END_VAR

VAR
	SERVICEOMKOPPLARE: fbManualOverride;

	UPPSTARTSSEKVENSIERING: BOOL;
END_VAR

VAR_OUTPUT
	bTILL:BOOL;

END_VAR
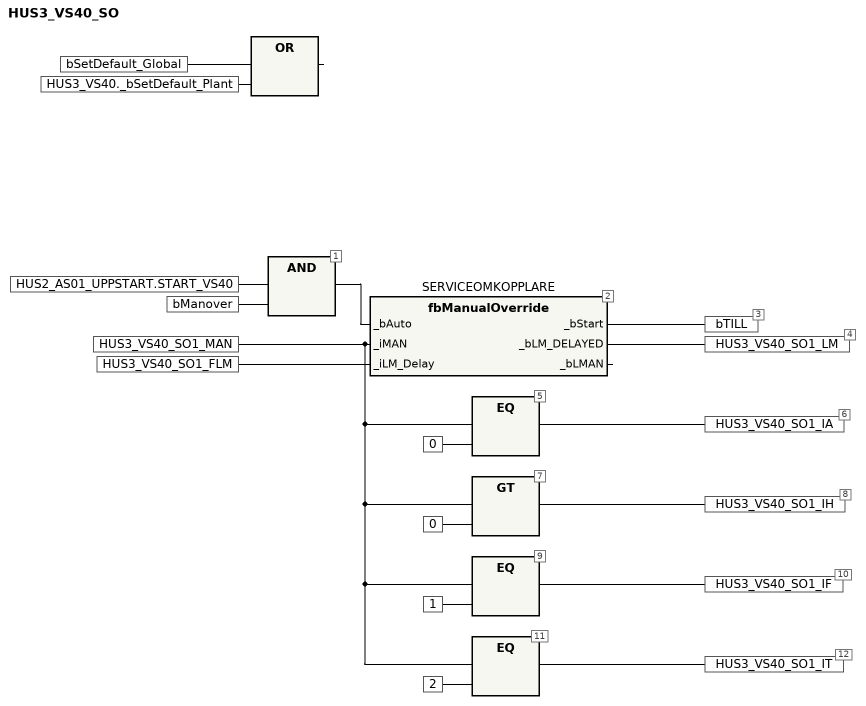
_CFC_ (* Continuous Function Chart, elements in execution order *)
#0 OR(bSetDefault_Global, HUS3_VS40._bSetDefault_Plant)
#1 AND(HUS2_AS01_UPPSTART.START_VS40, bManover)
#2 SERVICEOMKOPPLARE:fbManualOverride(_bAuto: #1, _iMAN: HUS3_VS40_SO1_MAN, _iLM_Delay: HUS3_VS40_SO1_FLM)
#3 bTILL <= #2._bStart
#4 HUS3_VS40_SO1_LM <= #2._bLM_DELAYED
#5 EQ(HUS3_VS40_SO1_MAN, 0)
#6 HUS3_VS40_SO1_IA <= #5
#7 GT(HUS3_VS40_SO1_MAN, 0)
#8 HUS3_VS40_SO1_IH <= #7
#9 EQ(HUS3_VS40_SO1_MAN, 1)
#10 HUS3_VS40_SO1_IF <= #9
#11 EQ(HUS3_VS40_SO1_MAN, 2)
#12 HUS3_VS40_SO1_IT <= #11
_END_CFC_
(* the same logic as Structured Text *)
(* result unused: bSetDefault_Global OR HUS3_VS40._bSetDefault_Plant *)
SERVICEOMKOPPLARE(_bAuto := HUS2_AS01_UPPSTART.START_VS40 AND bManover, _iMAN := HUS3_VS40_SO1_MAN, _iLM_Delay := HUS3_VS40_SO1_FLM);
bTILL := SERVICEOMKOPPLARE._bStart;
HUS3_VS40_SO1_LM := SERVICEOMKOPPLARE._bLM_DELAYED;
HUS3_VS40_SO1_IA := HUS3_VS40_SO1_MAN = 0;
HUS3_VS40_SO1_IH := HUS3_VS40_SO1_MAN > 0;
HUS3_VS40_SO1_IF := HUS3_VS40_SO1_MAN = 1;
HUS3_VS40_SO1_IT := HUS3_VS40_SO1_MAN = 2;
END_PROGRAM

(* POU SYSTEM/VS40/Pumpstyrning/HUS3_VS40_PV01, CFC *)
PROGRAM HUS3_VS40_PV01

VAR

	Default: BOOL;
	Motor: FB_HVACMotor1Speed;


	fbReset1: fbBool_Reset;
	AlarmDelay: fbDelayedAlarmSeconds;

	MANHAND: fbManualOverride;
END_VAR
VAR


(********************MOTOR********************)
(*INPUT*)
	eCtrlModeActuator			:E_HVACActuatorMode;
	tStartDelay						:TIME;
	tStopDelay						:TIME;
	tDelayFeedbContactor			:TIME:=T#30s;
	tFeedbProcessTimer				:TIME:=T#30s;
	tDelayFeedbProcess				:TIME:=T#30s;
(*OUTPUT*)
	byState							:BYTE ;
	bStateAuto							:BOOL;
	bStateRepairSwitch				:BOOL;
	bStateManSwitch				:BOOL;
	eStateModeActuator				:E_HVACActuatorMode;
	byError							:BYTE ;
	bErrorMotorprotec				:BOOL;
	bErrorFeedbContactor			:BOOL;
	bErrorFeedbProcess			:BOOL;
	bInvalidParameter				:BOOL;

END_VAR

VAR_INPUT
	_bAuto							:BOOL;(* enable function block *)
END_VAR

VAR_OUTPUT
	_bMANOVER						:BOOL;
	_bDRIFTFEL						:BOOL;
	_bLHAND							:BOOL;
END_VAR
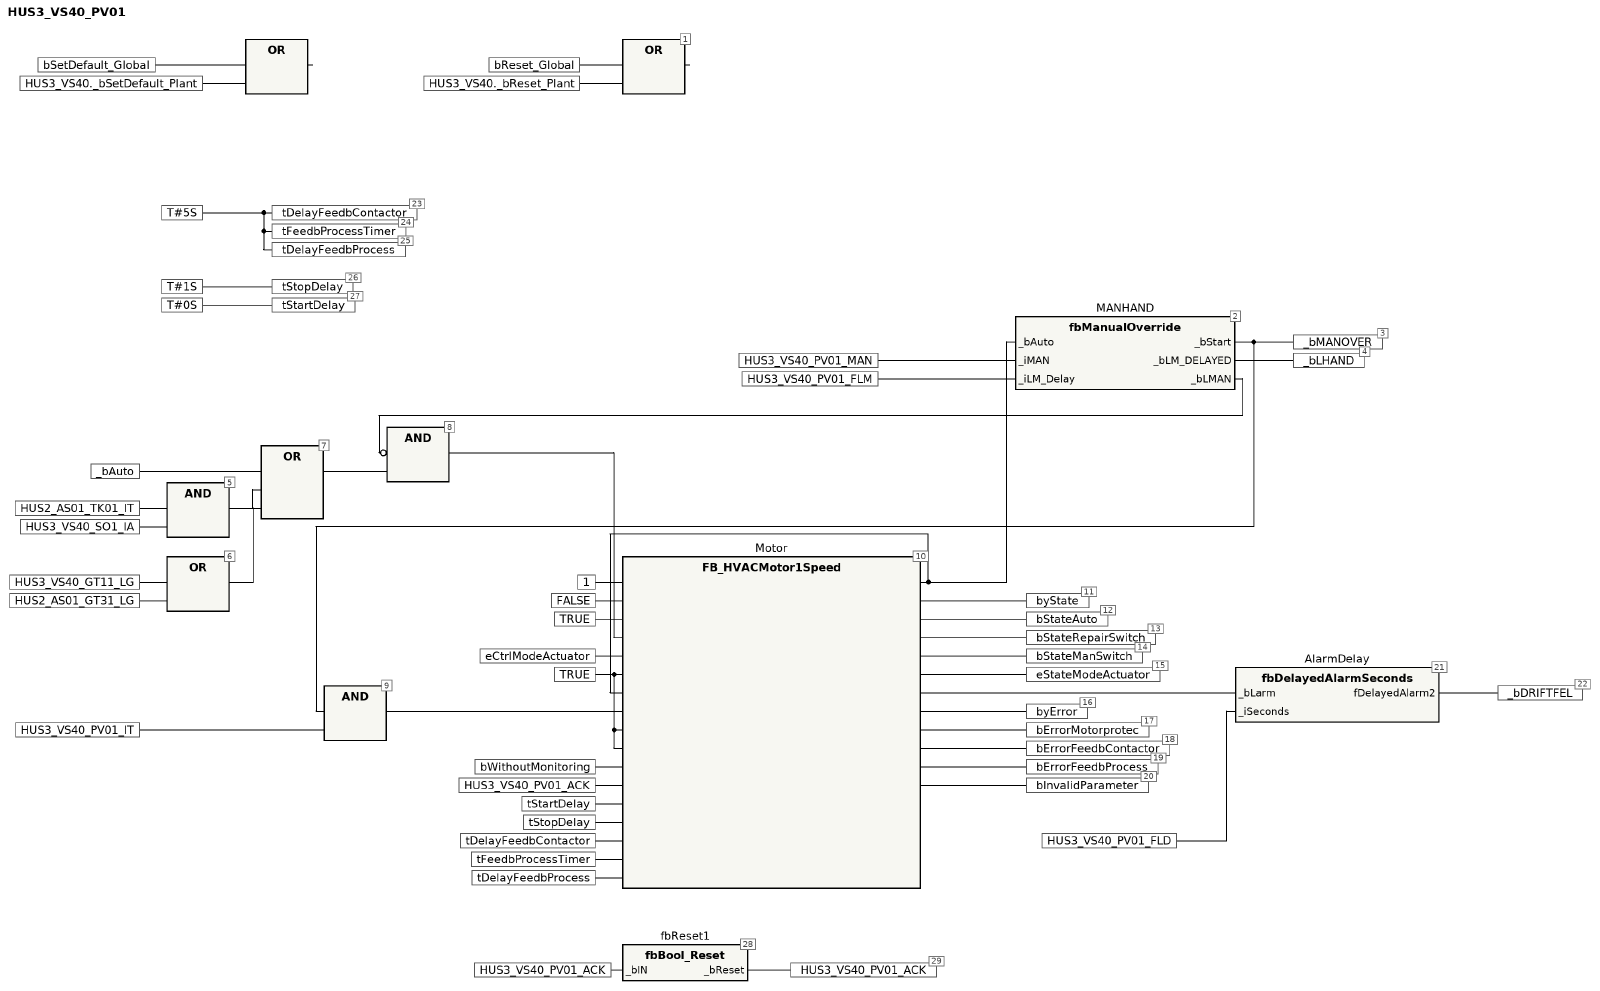
_CFC_ (* Continuous Function Chart, elements in execution order *)
#0 OR(bSetDefault_Global, HUS3_VS40._bSetDefault_Plant)
#1 OR(bReset_Global, HUS3_VS40._bReset_Plant)
#2 MANHAND:fbManualOverride(_bAuto: #10.out 1, _iMAN: HUS3_VS40_PV01_MAN, _iLM_Delay: HUS3_VS40_PV01_FLM)
#3 _bMANOVER <= #2._bStart
#4 _bLHAND <= #2._bLM_DELAYED
#5 AND(HUS2_AS01_TK01_IT, HUS3_VS40_SO1_IA)
#6 OR(HUS3_VS40_GT11_LG, HUS2_AS01_GT31_LG)
#7 OR(_bAuto, #5, #6)
#8 AND(NOT #2._bLMAN, #7)
#9 AND(#2._bStart, HUS3_VS40_PV01_IT)
#10 Motor:FB_HVACMotor1Speed(1, FALSE, TRUE, #8, eCtrlModeActuator, TRUE, #10.out 1, #9, TRUE, TRUE, bWithoutMonitoring, HUS3_VS40_PV01_ACK, tStartDelay, tStopDelay, tDelayFeedbContactor, tFeedbProcessTimer, tDelayFeedbProcess)
#11 byState <= #10.out 2
#12 bStateAuto <= #10.out 3
#13 bStateRepairSwitch <= #10.out 4
#14 bStateManSwitch <= #10.out 5
#15 eStateModeActuator <= #10.out 6
#16 byError <= #10.out 8
#17 bErrorMotorprotec <= #10.out 9
#18 bErrorFeedbContactor <= #10.out 10
#19 bErrorFeedbProcess <= #10.out 11
#20 bInvalidParameter <= #10.out 12
#21 AlarmDelay:fbDelayedAlarmSeconds(_bLarm: #10.out 7, _iSeconds: HUS3_VS40_PV01_FLD)
#22 _bDRIFTFEL <= #21.fDelayedAlarm2
#23 tDelayFeedbContactor <= T#5S
#24 tFeedbProcessTimer <= T#5S
#25 tDelayFeedbProcess <= T#5S
#26 tStopDelay <= T#1S
#27 tStartDelay <= T#0S
#28 fbReset1:fbBool_Reset(_bIN: HUS3_VS40_PV01_ACK)
#29 HUS3_VS40_PV01_ACK <= #28._bReset
_END_CFC_
END_PROGRAM

(* POU SYSTEM/VS40/Tempreglering/HUS3_VS40_GT11_PID, FAI *)
PROGRAM HUS3_VS40_GT11_PID

VAR_INPUT
	_bEnable		:BOOL;
	_rBV			:REAL;
	_rMV			:REAL;
END_VAR

VAR_OUTPUT
	_rY1                         : REAL;
END_VAR


VAR
	_bSetDefaultPID:BOOL;
	_bReset_Local:BOOL;


	SVX: FB_HVACPIDCtrl;
	eDataSecurityType         : E_HVACDataSecurityType;
	rInitialValue            : REAL;
	bResetController          : BOOL;
	_eCtrlMode				:E_HVACCtrlMode;(*
									eHVACCtrlMode_Auto      := 0,
								   	eHVACCtrlMode_Manual   := 1 *)
	_rOverrideValue			:REAL;(* controller output rY in operating mode eCtrlMode =1 *)
	rXW                        : REAL;
	bMaxLimit                  : BOOL;
	bMinLimit                  : BOOL;
	bActive                    : BOOL;
	bARWactive                 : BOOL;
	eState                     : E_HVACState;
	bError                     : BOOL;
	eErrorCode                 : E_HVACErrorCodes;
	bInvalidParameter          : BOOL;

	bDirection              : BOOL;
	_rKP: REAL;
	_rCH: REAL;
	tTi                     : TIME;
	tTv                     : TIME;
	tTd                     : TIME;

	rYMin                   : REAL;
	rYMax                   : REAL;

	CI: fbBer_PID_inst;
	CS: fbBer_PID_inst;
	CD: fbBer_PID_inst;

	fbPersistent_CH: FB_HVACPersistent_Real;
	fbPersistent_CP: FB_HVACPersistent_Real;
	fbPersistent_CI: FB_HVACPersistent_Real;
	fbPersistent_CS: FB_HVACPersistent_Real;
	fbPersistent_CD: FB_HVACPersistent_Real;
	LM_DELAY: fbDelayedAlarmMinutes;
END_VAR
(* body not read: cfc97 *)
END_PROGRAM

(* POU SYSTEM/VS40/Börvärden & kurvor/HUS3_VS40_GT11_KURVA, FAI *)
PROGRAM HUS3_VS40_GT11_KURVA
VAR
(****************************************** heating curve **********************************************************************************************************************)

	_bSetDefaultHC			:BOOL;


	fbScale_n:			FB_HVACScale_nPoint;
	_bErrParam:			BOOL;								(*ParameterError*)
	stScaleParameter:	ST_HVACParameterScale_nPoint	;	(*Parameter struktur på antal brutpunkter*)


	fbTemp1:	FB_HVACPersistent_Real;
	fbTemp2:	FB_HVACPersistent_Real;
	fbTemp3:	FB_HVACPersistent_Real;
	fbTemp4:	FB_HVACPersistent_Real;
	fbTemp5:	FB_HVACPersistent_Real;

	fbOutsideTemp1:	FB_HVACPersistent_Real;
	fbOutsideTemp2:	FB_HVACPersistent_Real;
	fbOutsideTemp3:	FB_HVACPersistent_Real;
	fbOutsideTemp4:	FB_HVACPersistent_Real;
	fbOutsideTemp5:	FB_HVACPersistent_Real;
	BB_min: FB_HVACPersistent_Real;
	BB_max: FB_HVACPersistent_Real;

END_VAR

VAR_INPUT
	_rGT3N	:REAL; (*Utegivare*)

END_VAR

VAR_OUTPUT
	_rBB		:LREAL;
END_VAR
(* body not read: cfc97 *)
END_PROGRAM

(* POU SYSTEM/VS40/Börvärden & kurvor/HUS3_VS40_EFFEKTBEGR, FAI *)
PROGRAM HUS3_VS40_EFFEKTBEGR
VAR
(****************************************** heating curve **********************************************************************************************************************)

	_bSetDefaultHC			:BOOL;


	fbScale_n:			FB_HVACScale_nPoint;
	_bErrParam:			BOOL;								(*ParameterError*)
	stScaleParameter:	ST_HVACParameterScale_nPoint	;	(*Parameter struktur på antal brutpunkter*)


	fbTemp1:	FB_HVACPersistent_Real;
	fbTemp2:	FB_HVACPersistent_Real;
	fbTemp3:	FB_HVACPersistent_Real;
	fbTemp4:	FB_HVACPersistent_Real;
	fbTemp5:	FB_HVACPersistent_Real;

	fbOutsideTemp1:	FB_HVACPersistent_Real;
	fbOutsideTemp2:	FB_HVACPersistent_Real;
	fbOutsideTemp3:	FB_HVACPersistent_Real;
	fbOutsideTemp4:	FB_HVACPersistent_Real;
	fbOutsideTemp5:	FB_HVACPersistent_Real;
	BB_min: FB_HVACPersistent_Real;
	BB_max: FB_HVACPersistent_Real;

	CalcForskjutning: fbConversionScale;

	MIN_LIMIT: REAL;
END_VAR

VAR_INPUT
	_rGT3N	:REAL; (*Utegivare*)
	_rMQ41_SV	:REAL;

END_VAR

VAR_OUTPUT
	_rBB		:LREAL;
END_VAR
(* body not read: cfc97 *)
END_PROGRAM

(* POU SYSTEM/VS40/Larm/HUS3_VS40_GT11_LARM, FAI *)
PROGRAM HUS3_VS40_GT11_LARM

VAR_OUTPUT
	_bLSumma					: BOOL;	(*Summalarm*)

END_VAR
VAR

	_bSetDefault: 				BOOL;		(*Se default values*)
	fbLarm: fbAvvikelselarm;


	fbHigh: FB_HVACPersistent_Real;
	fbAlarmDelayLH: FB_HVACPersistent_Int;
	fbLow: FB_HVACPersistent_Real;
	fbAlarmDelayLL: FB_HVACPersistent_Int;


END_VAR
(* body not read: cfc97 *)
END_PROGRAM

(* POU SYSTEM/FA101, FA102/HUS1_FA101_FA102, CFC *)
PROGRAM HUS1_FA101_FA102
VAR
	_bSetDefault_Plant		:BOOL;
	_bReset_Plant				:BOOL;

	HUS1_FA101_FF01_M: BOOL;
	HUS1_FA102_FF01_M: BOOL;

	OVERRIDE_FA101: fbManualOverrideAnalog;
	OVERRIDE_FA102: fbManualOverrideAnalog;

END_VAR
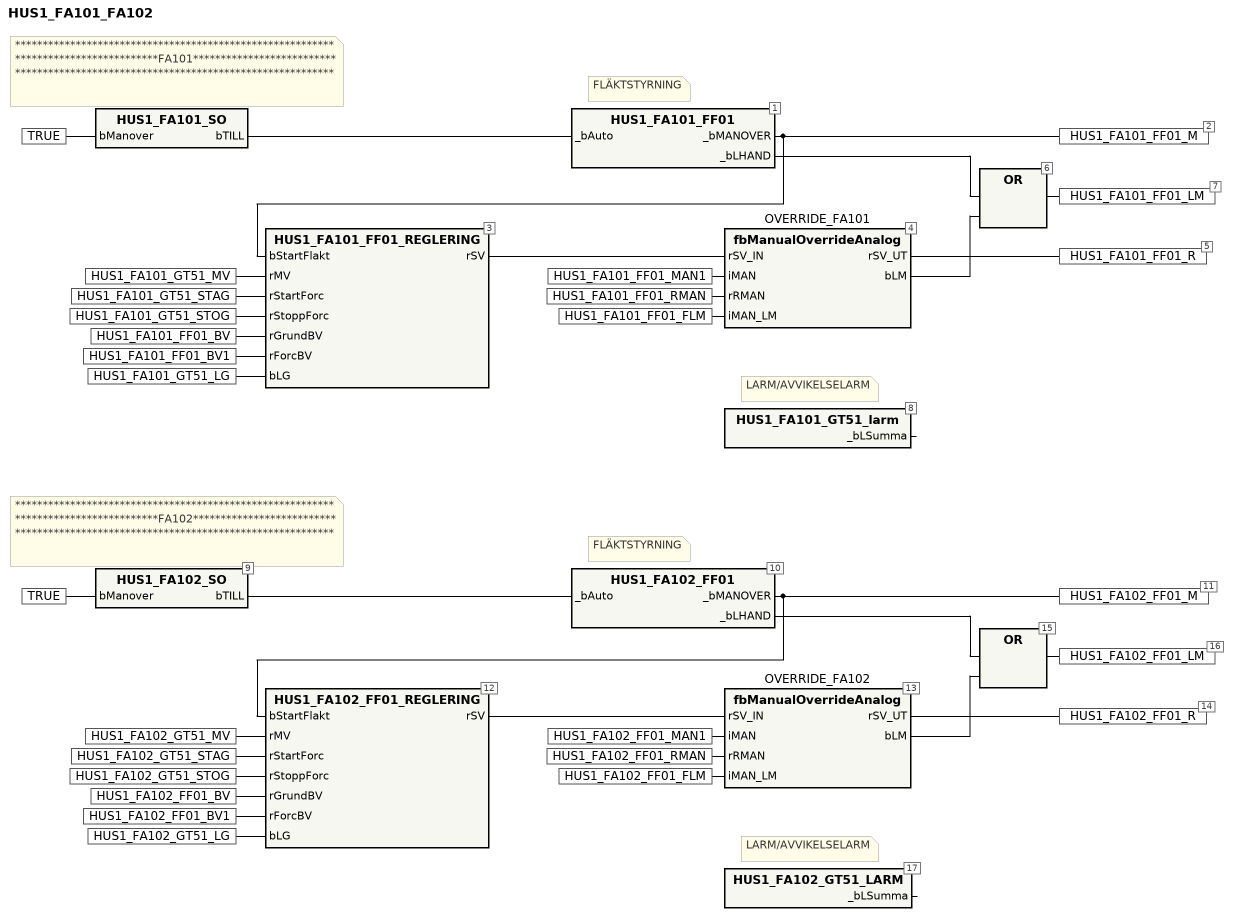
_CFC_ (* Continuous Function Chart, elements in execution order *)
(* ************************************************************************************FA101************************************************************************************ *)
(* ************************************************************************************FA102************************************************************************************ *)
(* FLÄKTSTYRNING *)
(* LARM/AVVIKELSELARM *)
(* FLÄKTSTYRNING *)
(* LARM/AVVIKELSELARM *)
#0 HUS1_FA101_SO(bManover: TRUE)
#1 HUS1_FA101_FF01(_bAuto: #0.bTILL)
#2 HUS1_FA101_FF01_M <= #1._bMANOVER
#3 HUS1_FA101_FF01_REGLERING(bStartFlakt: #1._bMANOVER, rMV: HUS1_FA101_GT51_MV, rStartForc: HUS1_FA101_GT51_STAG, rStoppForc: HUS1_FA101_GT51_STOG, rGrundBV: HUS1_FA101_FF01_BV, rForcBV: HUS1_FA101_FF01_BV1, bLG: HUS1_FA101_GT51_LG)
#4 OVERRIDE_FA101:fbManualOverrideAnalog(rSV_IN: #3.rSV, iMAN: HUS1_FA101_FF01_MAN1, rRMAN: HUS1_FA101_FF01_RMAN, iMAN_LM: HUS1_FA101_FF01_FLM)
#5 HUS1_FA101_FF01_R <= #4.rSV_UT
#6 OR(#1._bLHAND, #4.bLM)
#7 HUS1_FA101_FF01_LM <= #6
#8 HUS1_FA101_GT51_larm()
#9 HUS1_FA102_SO(bManover: TRUE)
#10 HUS1_FA102_FF01(_bAuto: #9.bTILL)
#11 HUS1_FA102_FF01_M <= #10._bMANOVER
#12 HUS1_FA102_FF01_REGLERING(bStartFlakt: #10._bMANOVER, rMV: HUS1_FA102_GT51_MV, rStartForc: HUS1_FA102_GT51_STAG, rStoppForc: HUS1_FA102_GT51_STOG, rGrundBV: HUS1_FA102_FF01_BV, rForcBV: HUS1_FA102_FF01_BV1, bLG: HUS1_FA102_GT51_LG)
#13 OVERRIDE_FA102:fbManualOverrideAnalog(rSV_IN: #12.rSV, iMAN: HUS1_FA102_FF01_MAN1, rRMAN: HUS1_FA102_FF01_RMAN, iMAN_LM: HUS1_FA102_FF01_FLM)
#14 HUS1_FA102_FF01_R <= #13.rSV_UT
#15 OR(#10._bLHAND, #13.bLM)
#16 HUS1_FA102_FF01_LM <= #15
#17 HUS1_FA102_GT51_LARM()
_END_CFC_
(* the same logic as Structured Text *)
(* ************************************************************************************FA101************************************************************************************ *)
(* ************************************************************************************FA102************************************************************************************ *)
(* FLÄKTSTYRNING *)
(* LARM/AVVIKELSELARM *)
(* FLÄKTSTYRNING *)
(* LARM/AVVIKELSELARM *)
HUS1_FA101_SO(bManover := TRUE);
HUS1_FA101_FF01(_bAuto := HUS1_FA101_SO.bTILL);
HUS1_FA101_FF01_M := HUS1_FA101_FF01._bMANOVER;
HUS1_FA101_FF01_REGLERING(bStartFlakt := HUS1_FA101_FF01._bMANOVER, rMV := HUS1_FA101_GT51_MV, rStartForc := HUS1_FA101_GT51_STAG, rStoppForc := HUS1_FA101_GT51_STOG, rGrundBV := HUS1_FA101_FF01_BV, rForcBV := HUS1_FA101_FF01_BV1, bLG := HUS1_FA101_GT51_LG);
OVERRIDE_FA101(rSV_IN := HUS1_FA101_FF01_REGLERING.rSV, iMAN := HUS1_FA101_FF01_MAN1, rRMAN := HUS1_FA101_FF01_RMAN, iMAN_LM := HUS1_FA101_FF01_FLM);
HUS1_FA101_FF01_R := OVERRIDE_FA101.rSV_UT;
HUS1_FA101_FF01_LM := HUS1_FA101_FF01._bLHAND OR OVERRIDE_FA101.bLM;
HUS1_FA101_GT51_larm();
HUS1_FA102_SO(bManover := TRUE);
HUS1_FA102_FF01(_bAuto := HUS1_FA102_SO.bTILL);
HUS1_FA102_FF01_M := HUS1_FA102_FF01._bMANOVER;
HUS1_FA102_FF01_REGLERING(bStartFlakt := HUS1_FA102_FF01._bMANOVER, rMV := HUS1_FA102_GT51_MV, rStartForc := HUS1_FA102_GT51_STAG, rStoppForc := HUS1_FA102_GT51_STOG, rGrundBV := HUS1_FA102_FF01_BV, rForcBV := HUS1_FA102_FF01_BV1, bLG := HUS1_FA102_GT51_LG);
OVERRIDE_FA102(rSV_IN := HUS1_FA102_FF01_REGLERING.rSV, iMAN := HUS1_FA102_FF01_MAN1, rRMAN := HUS1_FA102_FF01_RMAN, iMAN_LM := HUS1_FA102_FF01_FLM);
HUS1_FA102_FF01_R := OVERRIDE_FA102.rSV_UT;
HUS1_FA102_FF01_LM := HUS1_FA102_FF01._bLHAND OR OVERRIDE_FA102.bLM;
HUS1_FA102_GT51_LARM();
END_PROGRAM

(* POU xEgna Funktionsblock/fbManualOverrideAnalog, CFC *)
FUNCTION_BLOCK fbManualOverrideAnalog
VAR_INPUT
	rSV_IN			:REAL;
	iMAN			:INT;
	rRMAN		:REAL;
	iMAN_LM	:INT;

END_VAR
VAR_OUTPUT
	rSV_UT		:REAL;
	bLM		:BOOL;
END_VAR


VAR
	LM_DELAY: fbDelayedAlarmMinutes;
END_VAR
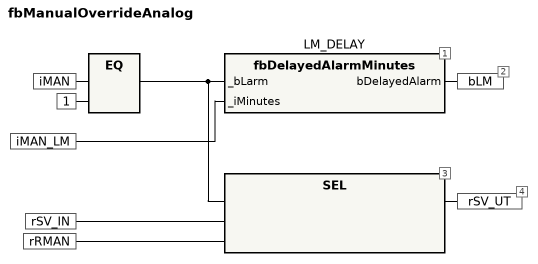
_CFC_ (* Continuous Function Chart, elements in execution order *)
#0 EQ(iMAN, 1)
#1 LM_DELAY:fbDelayedAlarmMinutes(_bLarm: #0, _iMinutes: iMAN_LM)
#2 bLM <= #1.bDelayedAlarm
#3 SEL(#0, rSV_IN, rRMAN)
#4 rSV_UT <= #3
_END_CFC_
END_FUNCTION_BLOCK

(* POU SYSTEM/FA101, FA102/HUS1_FA101_SO, CFC *)
PROGRAM HUS1_FA101_SO
VAR_INPUT

	bManover: BOOL;
END_VAR

VAR
	SERVICEOMKOPPLARE: fbManualOverride;

	UPPSTARTSSEKVENSIERING: BOOL;
END_VAR

VAR_OUTPUT
	bTILL:BOOL;

END_VAR
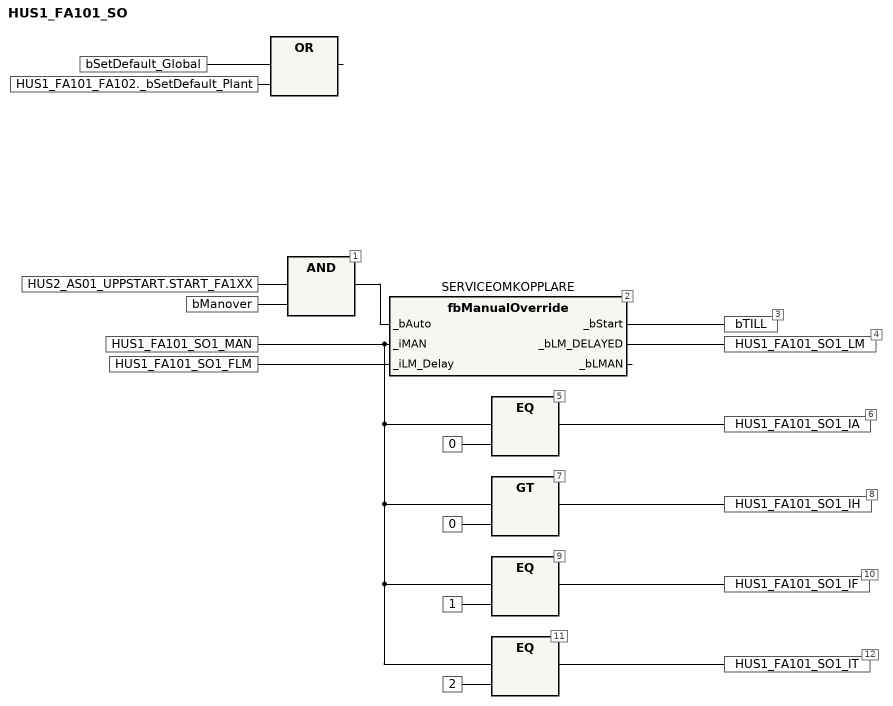
_CFC_ (* Continuous Function Chart, elements in execution order *)
#0 OR(bSetDefault_Global, HUS1_FA101_FA102._bSetDefault_Plant)
#1 AND(HUS2_AS01_UPPSTART.START_FA1XX, bManover)
#2 SERVICEOMKOPPLARE:fbManualOverride(_bAuto: #1, _iMAN: HUS1_FA101_SO1_MAN, _iLM_Delay: HUS1_FA101_SO1_FLM)
#3 bTILL <= #2._bStart
#4 HUS1_FA101_SO1_LM <= #2._bLM_DELAYED
#5 EQ(HUS1_FA101_SO1_MAN, 0)
#6 HUS1_FA101_SO1_IA <= #5
#7 GT(HUS1_FA101_SO1_MAN, 0)
#8 HUS1_FA101_SO1_IH <= #7
#9 EQ(HUS1_FA101_SO1_MAN, 1)
#10 HUS1_FA101_SO1_IF <= #9
#11 EQ(HUS1_FA101_SO1_MAN, 2)
#12 HUS1_FA101_SO1_IT <= #11
_END_CFC_
(* the same logic as Structured Text *)
(* result unused: bSetDefault_Global OR HUS1_FA101_FA102._bSetDefault_Plant *)
SERVICEOMKOPPLARE(_bAuto := HUS2_AS01_UPPSTART.START_FA1XX AND bManover, _iMAN := HUS1_FA101_SO1_MAN, _iLM_Delay := HUS1_FA101_SO1_FLM);
bTILL := SERVICEOMKOPPLARE._bStart;
HUS1_FA101_SO1_LM := SERVICEOMKOPPLARE._bLM_DELAYED;
HUS1_FA101_SO1_IA := HUS1_FA101_SO1_MAN = 0;
HUS1_FA101_SO1_IH := HUS1_FA101_SO1_MAN > 0;
HUS1_FA101_SO1_IF := HUS1_FA101_SO1_MAN = 1;
HUS1_FA101_SO1_IT := HUS1_FA101_SO1_MAN = 2;
END_PROGRAM

(* POU SYSTEM/FA101, FA102/Fläktstyr/HUS1_FA101_FF01, CFC *)
PROGRAM HUS1_FA101_FF01

VAR
	MANHAND: fbManualOverride;





END_VAR
VAR

END_VAR

VAR_INPUT
	_bAuto							:BOOL;(* enable function block *)
END_VAR

VAR_OUTPUT
	_bMANOVER						:BOOL;
	_bLHAND							:BOOL;
END_VAR
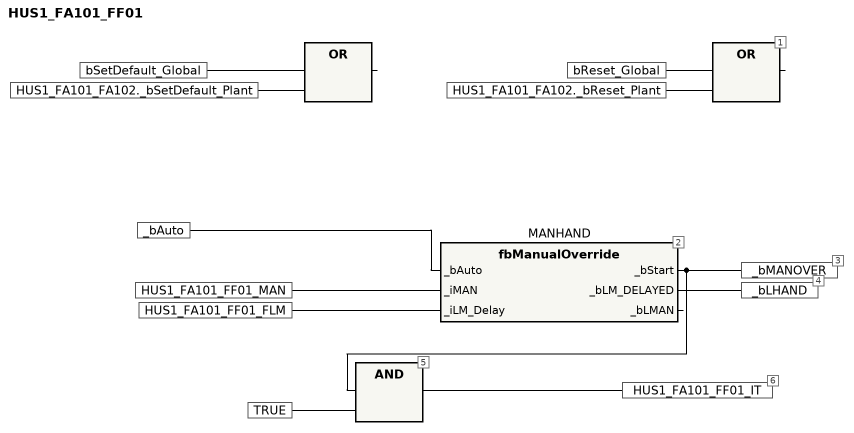
_CFC_ (* Continuous Function Chart, elements in execution order *)
#0 OR(bSetDefault_Global, HUS1_FA101_FA102._bSetDefault_Plant)
#1 OR(bReset_Global, HUS1_FA101_FA102._bReset_Plant)
#2 MANHAND:fbManualOverride(_bAuto: _bAuto, _iMAN: HUS1_FA101_FF01_MAN, _iLM_Delay: HUS1_FA101_FF01_FLM)
#3 _bMANOVER <= #2._bStart
#4 _bLHAND <= #2._bLM_DELAYED
#5 AND(#2._bStart, TRUE)
#6 HUS1_FA101_FF01_IT <= #5
_END_CFC_
(* the same logic as Structured Text *)
(* result unused: bSetDefault_Global OR HUS1_FA101_FA102._bSetDefault_Plant *)
(* result unused: bReset_Global OR HUS1_FA101_FA102._bReset_Plant *)
MANHAND(_bAuto := _bAuto, _iMAN := HUS1_FA101_FF01_MAN, _iLM_Delay := HUS1_FA101_FF01_FLM);
_bMANOVER := MANHAND._bStart;
_bLHAND := MANHAND._bLM_DELAYED;
HUS1_FA101_FF01_IT := MANHAND._bStart AND TRUE;
END_PROGRAM

(* POU SYSTEM/FA101, FA102/Fläktstyr/HUS1_FA101_FF01_REGLERING, CFC *)
PROGRAM HUS1_FA101_FF01_REGLERING

VAR
	SETRESET: SR;
END_VAR

VAR_INPUT
	bStartFlakt			:BOOL;
	rMV				:REAL;
	rStartForc			:REAL;
	rStoppForc		:REAL;
	rGrundBV			:REAL;
	rForcBV			:REAL;
	bLG				:BOOL;

END_VAR

VAR_OUTPUT
	rSV			:REAL;

END_VAR
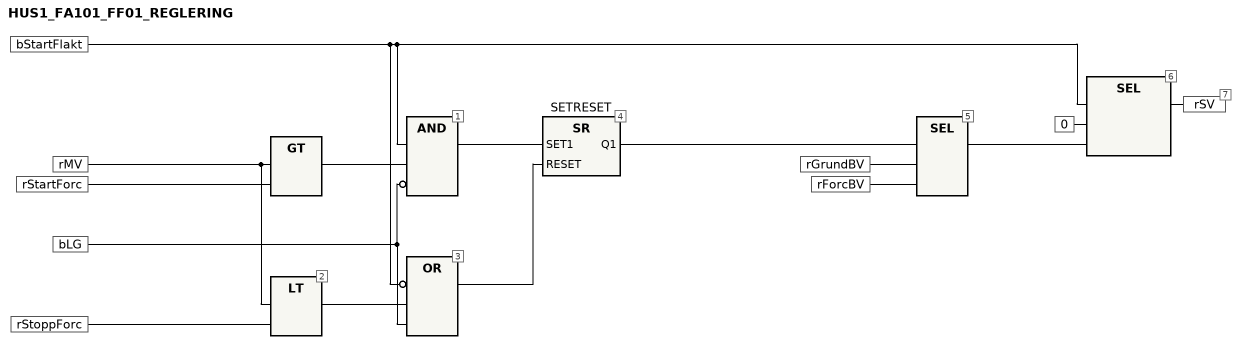
_CFC_ (* Continuous Function Chart, elements in execution order *)
#0 GT(rMV, rStartForc)
#1 AND(bStartFlakt, #0, NOT bLG)
#2 LT(rMV, rStoppForc)
#3 OR(NOT bStartFlakt, #2, bLG)
#4 SETRESET:SR(SET1: #1, RESET: #3)
#5 SEL(#4.Q1, rGrundBV, rForcBV)
#6 SEL(bStartFlakt, 0, #5)
#7 rSV <= #6
_END_CFC_
(* the same logic as Structured Text *)
SETRESET(SET1 := bStartFlakt AND (rMV > rStartForc) AND NOT bLG, RESET := NOT bStartFlakt OR (rMV < rStoppForc) OR bLG);
rSV := SEL(bStartFlakt, 0, SEL(SETRESET.Q1, rGrundBV, rForcBV));
END_PROGRAM

(* POU SYSTEM/FA101, FA102/Larm/HUS1_FA101_GT51_LARM, FAI *)
PROGRAM HUS1_FA101_GT51_LARM

VAR_OUTPUT
	_bLSumma					: BOOL;	(*Summalarm*)

END_VAR
VAR

	_bSetDefault: 				BOOL;		(*Se default values*)
	fbLarm: fbAvvikelselarm;


	fbHigh: FB_HVACPersistent_Real;
	fbAlarmDelayLH: FB_HVACPersistent_Int;


END_VAR
(* body not read: cfc97 *)
END_PROGRAM

(* POU SYSTEM/FA101, FA102/HUS1_FA102_SO, CFC *)
PROGRAM HUS1_FA102_SO
VAR_INPUT

	bManover: BOOL;
END_VAR

VAR
	SERVICEOMKOPPLARE: fbManualOverride;

	UPPSTARTSSEKVENSIERING: BOOL;
END_VAR

VAR_OUTPUT
	bTILL:BOOL;

END_VAR
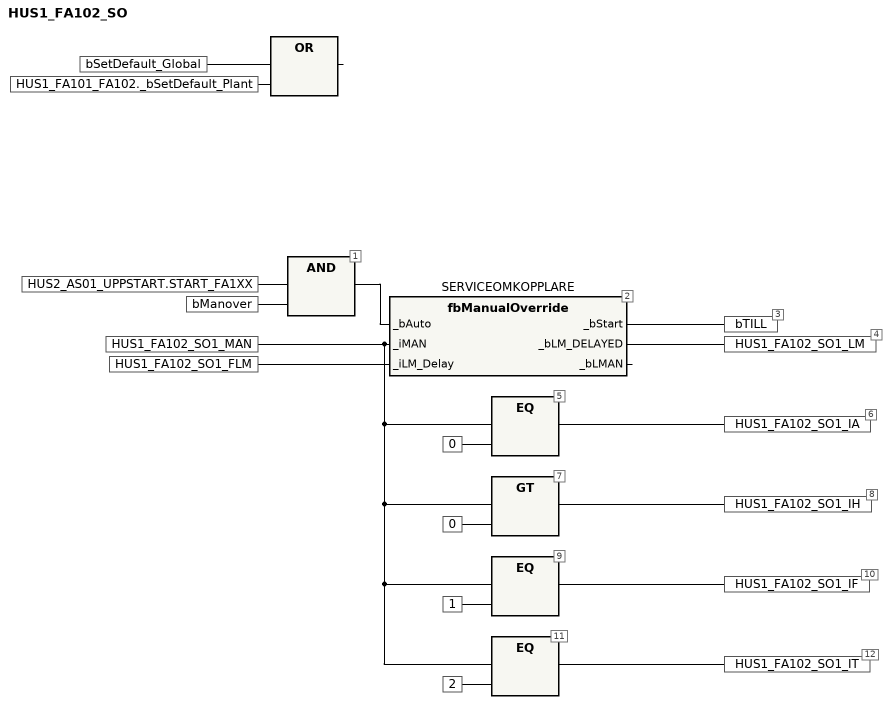
_CFC_ (* Continuous Function Chart, elements in execution order *)
#0 OR(bSetDefault_Global, HUS1_FA101_FA102._bSetDefault_Plant)
#1 AND(HUS2_AS01_UPPSTART.START_FA1XX, bManover)
#2 SERVICEOMKOPPLARE:fbManualOverride(_bAuto: #1, _iMAN: HUS1_FA102_SO1_MAN, _iLM_Delay: HUS1_FA102_SO1_FLM)
#3 bTILL <= #2._bStart
#4 HUS1_FA102_SO1_LM <= #2._bLM_DELAYED
#5 EQ(HUS1_FA102_SO1_MAN, 0)
#6 HUS1_FA102_SO1_IA <= #5
#7 GT(HUS1_FA102_SO1_MAN, 0)
#8 HUS1_FA102_SO1_IH <= #7
#9 EQ(HUS1_FA102_SO1_MAN, 1)
#10 HUS1_FA102_SO1_IF <= #9
#11 EQ(HUS1_FA102_SO1_MAN, 2)
#12 HUS1_FA102_SO1_IT <= #11
_END_CFC_
(* the same logic as Structured Text *)
(* result unused: bSetDefault_Global OR HUS1_FA101_FA102._bSetDefault_Plant *)
SERVICEOMKOPPLARE(_bAuto := HUS2_AS01_UPPSTART.START_FA1XX AND bManover, _iMAN := HUS1_FA102_SO1_MAN, _iLM_Delay := HUS1_FA102_SO1_FLM);
bTILL := SERVICEOMKOPPLARE._bStart;
HUS1_FA102_SO1_LM := SERVICEOMKOPPLARE._bLM_DELAYED;
HUS1_FA102_SO1_IA := HUS1_FA102_SO1_MAN = 0;
HUS1_FA102_SO1_IH := HUS1_FA102_SO1_MAN > 0;
HUS1_FA102_SO1_IF := HUS1_FA102_SO1_MAN = 1;
HUS1_FA102_SO1_IT := HUS1_FA102_SO1_MAN = 2;
END_PROGRAM

(* POU SYSTEM/FA101, FA102/Fläktstyr/HUS1_FA102_FF01, CFC *)
PROGRAM HUS1_FA102_FF01

VAR
	MANHAND: fbManualOverride;





END_VAR
VAR

END_VAR

VAR_INPUT
	_bAuto							:BOOL;(* enable function block *)
END_VAR

VAR_OUTPUT
	_bMANOVER						:BOOL;
	_bLHAND							:BOOL;
END_VAR
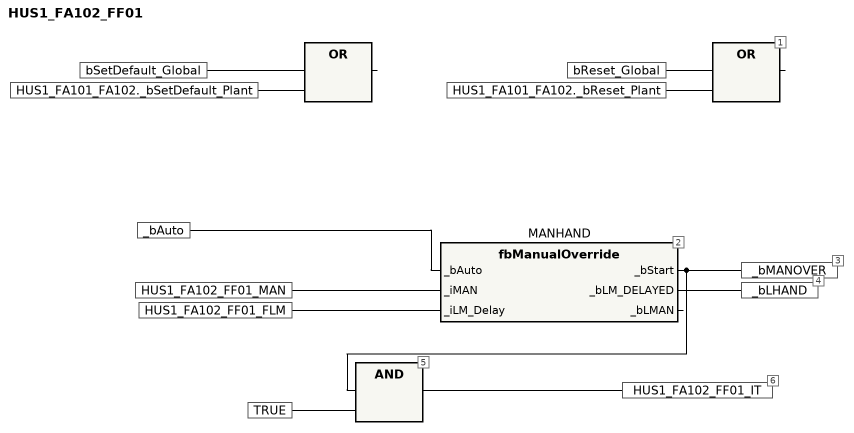
_CFC_ (* Continuous Function Chart, elements in execution order *)
#0 OR(bSetDefault_Global, HUS1_FA101_FA102._bSetDefault_Plant)
#1 OR(bReset_Global, HUS1_FA101_FA102._bReset_Plant)
#2 MANHAND:fbManualOverride(_bAuto: _bAuto, _iMAN: HUS1_FA102_FF01_MAN, _iLM_Delay: HUS1_FA102_FF01_FLM)
#3 _bMANOVER <= #2._bStart
#4 _bLHAND <= #2._bLM_DELAYED
#5 AND(#2._bStart, TRUE)
#6 HUS1_FA102_FF01_IT <= #5
_END_CFC_
(* the same logic as Structured Text *)
(* result unused: bSetDefault_Global OR HUS1_FA101_FA102._bSetDefault_Plant *)
(* result unused: bReset_Global OR HUS1_FA101_FA102._bReset_Plant *)
MANHAND(_bAuto := _bAuto, _iMAN := HUS1_FA102_FF01_MAN, _iLM_Delay := HUS1_FA102_FF01_FLM);
_bMANOVER := MANHAND._bStart;
_bLHAND := MANHAND._bLM_DELAYED;
HUS1_FA102_FF01_IT := MANHAND._bStart AND TRUE;
END_PROGRAM

(* POU SYSTEM/FA101, FA102/Fläktstyr/HUS1_FA102_FF01_REGLERING, CFC *)
PROGRAM HUS1_FA102_FF01_REGLERING

VAR
	SETRESET: SR;
END_VAR

VAR_INPUT
	bStartFlakt			:BOOL;
	rMV				:REAL;
	rStartForc			:REAL;
	rStoppForc		:REAL;
	rGrundBV			:REAL;
	rForcBV			:REAL;
	bLG				:BOOL;

END_VAR

VAR_OUTPUT
	rSV			:REAL;

END_VAR
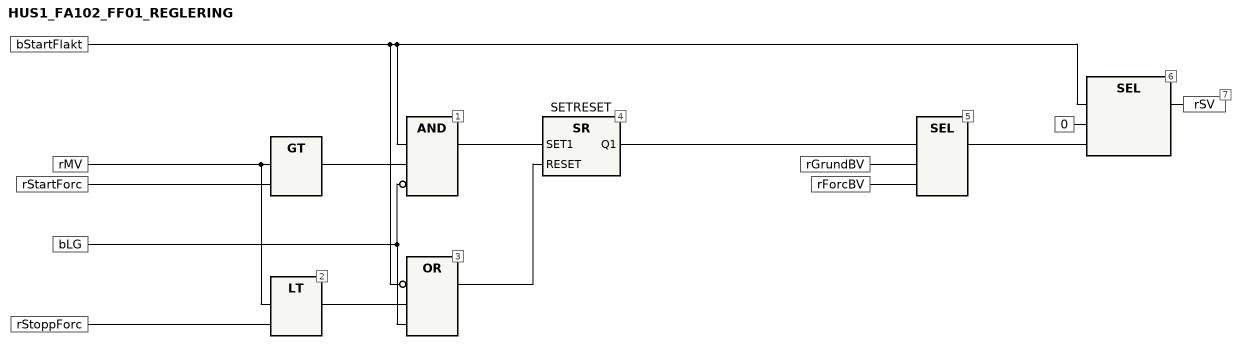
_CFC_ (* Continuous Function Chart, elements in execution order *)
#0 GT(rMV, rStartForc)
#1 AND(bStartFlakt, #0, NOT bLG)
#2 LT(rMV, rStoppForc)
#3 OR(NOT bStartFlakt, #2, bLG)
#4 SETRESET:SR(SET1: #1, RESET: #3)
#5 SEL(#4.Q1, rGrundBV, rForcBV)
#6 SEL(bStartFlakt, 0, #5)
#7 rSV <= #6
_END_CFC_
(* the same logic as Structured Text *)
SETRESET(SET1 := bStartFlakt AND (rMV > rStartForc) AND NOT bLG, RESET := NOT bStartFlakt OR (rMV < rStoppForc) OR bLG);
rSV := SEL(bStartFlakt, 0, SEL(SETRESET.Q1, rGrundBV, rForcBV));
END_PROGRAM

(* POU SYSTEM/FA101, FA102/Larm/HUS1_FA102_GT51_LARM, FAI *)
PROGRAM HUS1_FA102_GT51_LARM

VAR_OUTPUT
	_bLSumma					: BOOL;	(*Summalarm*)

END_VAR
VAR

	_bSetDefault: 				BOOL;		(*Se default values*)
	fbLarm: fbAvvikelselarm;


	fbHigh: FB_HVACPersistent_Real;
	fbAlarmDelayLH: FB_HVACPersistent_Int;


END_VAR
(* body not read: cfc97 *)
END_PROGRAM

(* POU SYSTEM/FA201, FA202, FA203/HUS2_FA201_FA203, CFC *)
PROGRAM HUS2_FA201_FA203
VAR
	_bSetDefault_Plant		:BOOL;
	_bReset_Plant				:BOOL;


	OVERRIDE_FA201: fbManualOverrideAnalog;
	OVERRIDE_FA202: fbManualOverrideAnalog;
	OVERRIDE_FA203: fbManualOverrideAnalog;
END_VAR
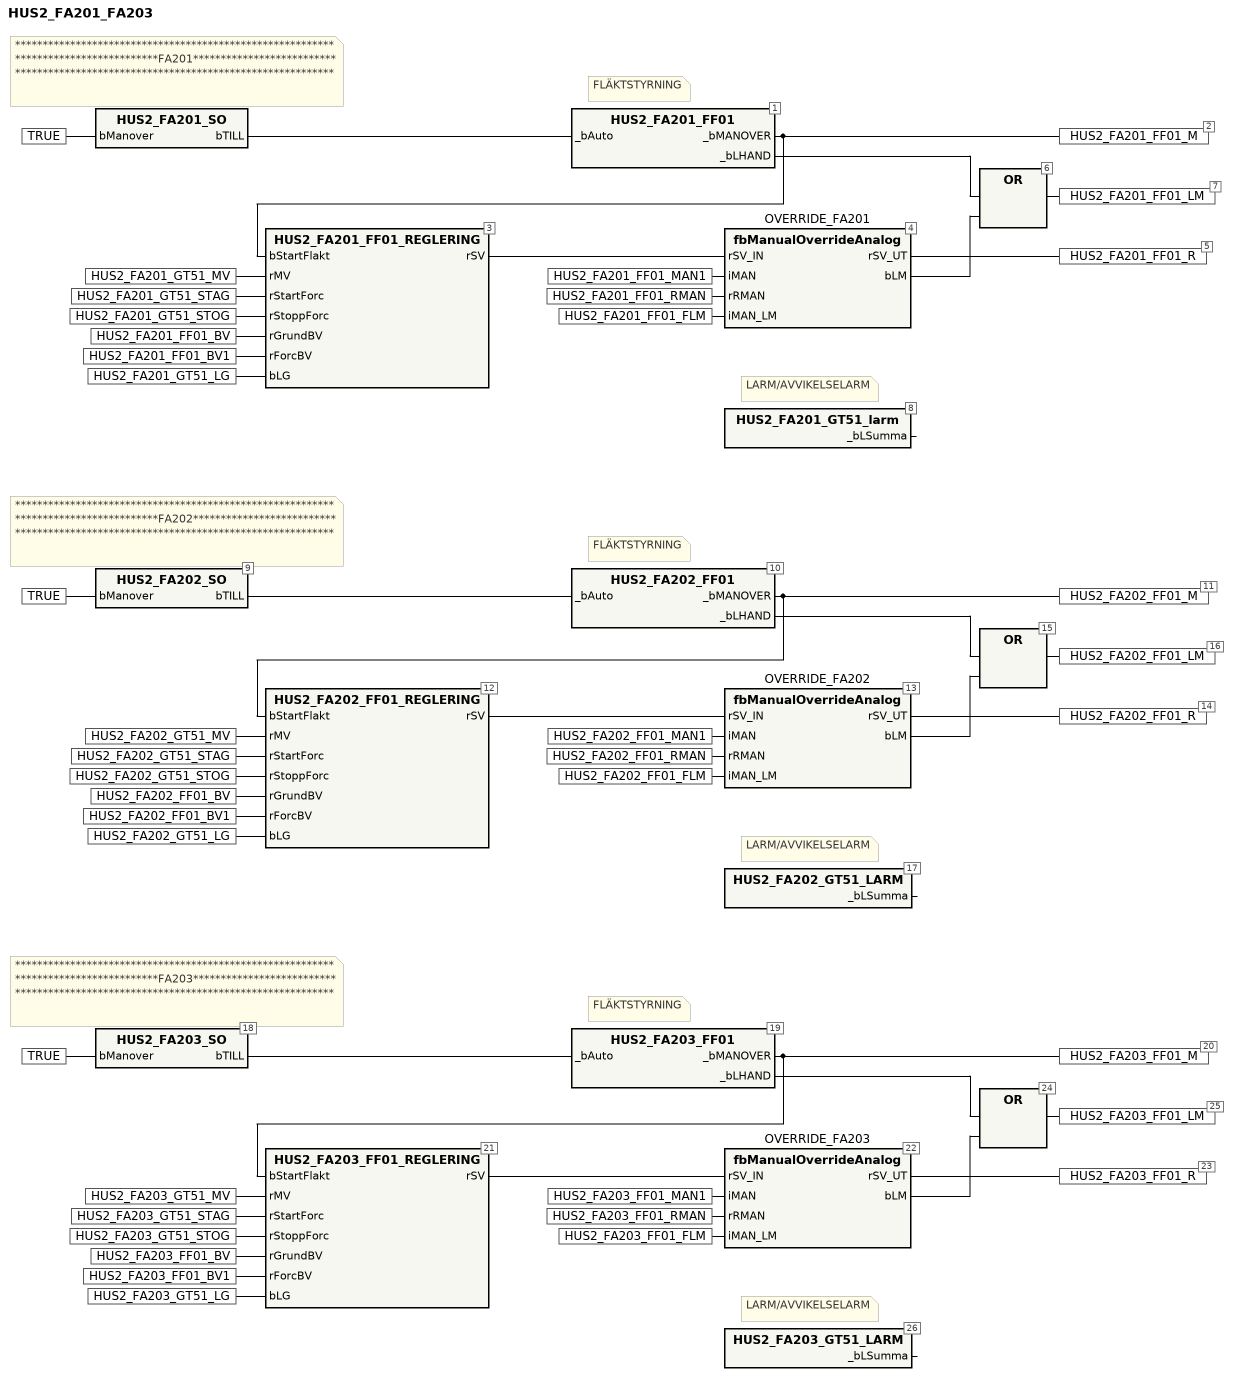
_CFC_ (* Continuous Function Chart, elements in execution order *)
(* LARM/AVVIKELSELARM *)
(* FLÄKTSTYRNING *)
(* ************************************************************************************FA203************************************************************************************ *)
(* LARM/AVVIKELSELARM *)
(* FLÄKTSTYRNING *)
(* LARM/AVVIKELSELARM *)
(* FLÄKTSTYRNING *)
(* ************************************************************************************FA202************************************************************************************ *)
(* ************************************************************************************FA201************************************************************************************ *)
#0 HUS2_FA201_SO(bManover: TRUE)
#1 HUS2_FA201_FF01(_bAuto: #0.bTILL)
#2 HUS2_FA201_FF01_M <= #1._bMANOVER
#3 HUS2_FA201_FF01_REGLERING(bStartFlakt: #1._bMANOVER, rMV: HUS2_FA201_GT51_MV, rStartForc: HUS2_FA201_GT51_STAG, rStoppForc: HUS2_FA201_GT51_STOG, rGrundBV: HUS2_FA201_FF01_BV, rForcBV: HUS2_FA201_FF01_BV1, bLG: HUS2_FA201_GT51_LG)
#4 OVERRIDE_FA201:fbManualOverrideAnalog(rSV_IN: #3.rSV, iMAN: HUS2_FA201_FF01_MAN1, rRMAN: HUS2_FA201_FF01_RMAN, iMAN_LM: HUS2_FA201_FF01_FLM)
#5 HUS2_FA201_FF01_R <= #4.rSV_UT
#6 OR(#1._bLHAND, #4.bLM)
#7 HUS2_FA201_FF01_LM <= #6
#8 HUS2_FA201_GT51_larm()
#9 HUS2_FA202_SO(bManover: TRUE)
#10 HUS2_FA202_FF01(_bAuto: #9.bTILL)
#11 HUS2_FA202_FF01_M <= #10._bMANOVER
#12 HUS2_FA202_FF01_REGLERING(bStartFlakt: #10._bMANOVER, rMV: HUS2_FA202_GT51_MV, rStartForc: HUS2_FA202_GT51_STAG, rStoppForc: HUS2_FA202_GT51_STOG, rGrundBV: HUS2_FA202_FF01_BV, rForcBV: HUS2_FA202_FF01_BV1, bLG: HUS2_FA202_GT51_LG)
#13 OVERRIDE_FA202:fbManualOverrideAnalog(rSV_IN: #12.rSV, iMAN: HUS2_FA202_FF01_MAN1, rRMAN: HUS2_FA202_FF01_RMAN, iMAN_LM: HUS2_FA202_FF01_FLM)
#14 HUS2_FA202_FF01_R <= #13.rSV_UT
#15 OR(#10._bLHAND, #13.bLM)
#16 HUS2_FA202_FF01_LM <= #15
#17 HUS2_FA202_GT51_LARM()
#18 HUS2_FA203_SO(bManover: TRUE)
#19 HUS2_FA203_FF01(_bAuto: #18.bTILL)
#20 HUS2_FA203_FF01_M <= #19._bMANOVER
#21 HUS2_FA203_FF01_REGLERING(bStartFlakt: #19._bMANOVER, rMV: HUS2_FA203_GT51_MV, rStartForc: HUS2_FA203_GT51_STAG, rStoppForc: HUS2_FA203_GT51_STOG, rGrundBV: HUS2_FA203_FF01_BV, rForcBV: HUS2_FA203_FF01_BV1, bLG: HUS2_FA203_GT51_LG)
#22 OVERRIDE_FA203:fbManualOverrideAnalog(rSV_IN: #21.rSV, iMAN: HUS2_FA203_FF01_MAN1, rRMAN: HUS2_FA203_FF01_RMAN, iMAN_LM: HUS2_FA203_FF01_FLM)
#23 HUS2_FA203_FF01_R <= #22.rSV_UT
#24 OR(#19._bLHAND, #22.bLM)
#25 HUS2_FA203_FF01_LM <= #24
#26 HUS2_FA203_GT51_LARM()
_END_CFC_
(* the same logic as Structured Text *)
(* LARM/AVVIKELSELARM *)
(* FLÄKTSTYRNING *)
(* ************************************************************************************FA203************************************************************************************ *)
(* LARM/AVVIKELSELARM *)
(* FLÄKTSTYRNING *)
(* LARM/AVVIKELSELARM *)
(* FLÄKTSTYRNING *)
(* ************************************************************************************FA202************************************************************************************ *)
(* ************************************************************************************FA201************************************************************************************ *)
HUS2_FA201_SO(bManover := TRUE);
HUS2_FA201_FF01(_bAuto := HUS2_FA201_SO.bTILL);
HUS2_FA201_FF01_M := HUS2_FA201_FF01._bMANOVER;
HUS2_FA201_FF01_REGLERING(bStartFlakt := HUS2_FA201_FF01._bMANOVER, rMV := HUS2_FA201_GT51_MV, rStartForc := HUS2_FA201_GT51_STAG, rStoppForc := HUS2_FA201_GT51_STOG, rGrundBV := HUS2_FA201_FF01_BV, rForcBV := HUS2_FA201_FF01_BV1, bLG := HUS2_FA201_GT51_LG);
OVERRIDE_FA201(rSV_IN := HUS2_FA201_FF01_REGLERING.rSV, iMAN := HUS2_FA201_FF01_MAN1, rRMAN := HUS2_FA201_FF01_RMAN, iMAN_LM := HUS2_FA201_FF01_FLM);
HUS2_FA201_FF01_R := OVERRIDE_FA201.rSV_UT;
HUS2_FA201_FF01_LM := HUS2_FA201_FF01._bLHAND OR OVERRIDE_FA201.bLM;
HUS2_FA201_GT51_larm();
HUS2_FA202_SO(bManover := TRUE);
HUS2_FA202_FF01(_bAuto := HUS2_FA202_SO.bTILL);
HUS2_FA202_FF01_M := HUS2_FA202_FF01._bMANOVER;
HUS2_FA202_FF01_REGLERING(bStartFlakt := HUS2_FA202_FF01._bMANOVER, rMV := HUS2_FA202_GT51_MV, rStartForc := HUS2_FA202_GT51_STAG, rStoppForc := HUS2_FA202_GT51_STOG, rGrundBV := HUS2_FA202_FF01_BV, rForcBV := HUS2_FA202_FF01_BV1, bLG := HUS2_FA202_GT51_LG);
OVERRIDE_FA202(rSV_IN := HUS2_FA202_FF01_REGLERING.rSV, iMAN := HUS2_FA202_FF01_MAN1, rRMAN := HUS2_FA202_FF01_RMAN, iMAN_LM := HUS2_FA202_FF01_FLM);
HUS2_FA202_FF01_R := OVERRIDE_FA202.rSV_UT;
HUS2_FA202_FF01_LM := HUS2_FA202_FF01._bLHAND OR OVERRIDE_FA202.bLM;
HUS2_FA202_GT51_LARM();
HUS2_FA203_SO(bManover := TRUE);
HUS2_FA203_FF01(_bAuto := HUS2_FA203_SO.bTILL);
HUS2_FA203_FF01_M := HUS2_FA203_FF01._bMANOVER;
HUS2_FA203_FF01_REGLERING(bStartFlakt := HUS2_FA203_FF01._bMANOVER, rMV := HUS2_FA203_GT51_MV, rStartForc := HUS2_FA203_GT51_STAG, rStoppForc := HUS2_FA203_GT51_STOG, rGrundBV := HUS2_FA203_FF01_BV, rForcBV := HUS2_FA203_FF01_BV1, bLG := HUS2_FA203_GT51_LG);
OVERRIDE_FA203(rSV_IN := HUS2_FA203_FF01_REGLERING.rSV, iMAN := HUS2_FA203_FF01_MAN1, rRMAN := HUS2_FA203_FF01_RMAN, iMAN_LM := HUS2_FA203_FF01_FLM);
HUS2_FA203_FF01_R := OVERRIDE_FA203.rSV_UT;
HUS2_FA203_FF01_LM := HUS2_FA203_FF01._bLHAND OR OVERRIDE_FA203.bLM;
HUS2_FA203_GT51_LARM();
END_PROGRAM

(* POU SYSTEM/FA201, FA202, FA203/HUS2_FA201_SO, CFC *)
PROGRAM HUS2_FA201_SO
VAR_INPUT

	bManover: BOOL;
END_VAR

VAR
	SERVICEOMKOPPLARE: fbManualOverride;

	UPPSTARTSSEKVENSIERING: BOOL;
END_VAR

VAR_OUTPUT
	bTILL:BOOL;

END_VAR
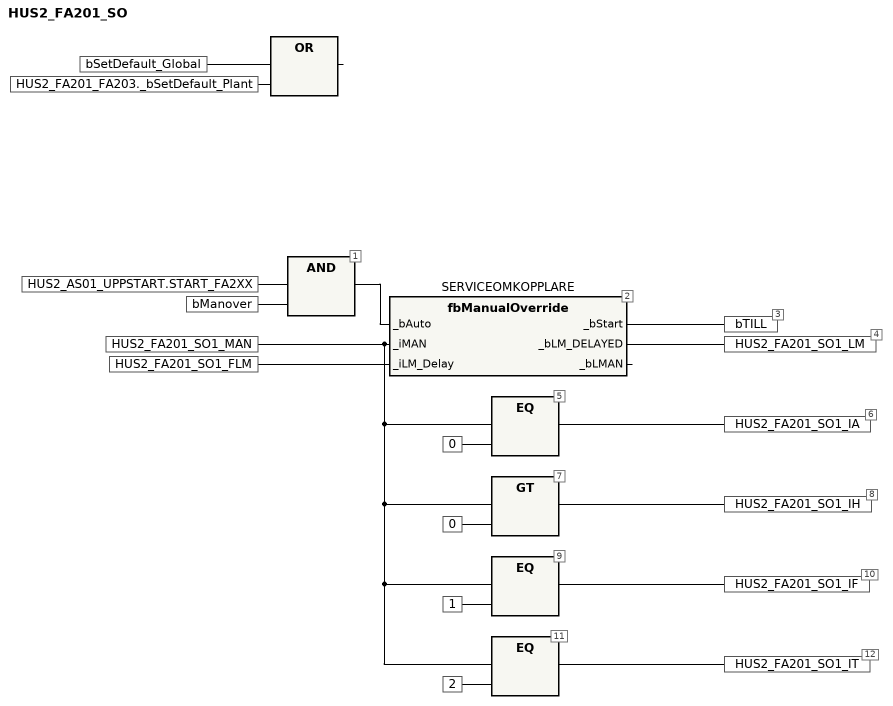
_CFC_ (* Continuous Function Chart, elements in execution order *)
#0 OR(bSetDefault_Global, HUS2_FA201_FA203._bSetDefault_Plant)
#1 AND(HUS2_AS01_UPPSTART.START_FA2XX, bManover)
#2 SERVICEOMKOPPLARE:fbManualOverride(_bAuto: #1, _iMAN: HUS2_FA201_SO1_MAN, _iLM_Delay: HUS2_FA201_SO1_FLM)
#3 bTILL <= #2._bStart
#4 HUS2_FA201_SO1_LM <= #2._bLM_DELAYED
#5 EQ(HUS2_FA201_SO1_MAN, 0)
#6 HUS2_FA201_SO1_IA <= #5
#7 GT(HUS2_FA201_SO1_MAN, 0)
#8 HUS2_FA201_SO1_IH <= #7
#9 EQ(HUS2_FA201_SO1_MAN, 1)
#10 HUS2_FA201_SO1_IF <= #9
#11 EQ(HUS2_FA201_SO1_MAN, 2)
#12 HUS2_FA201_SO1_IT <= #11
_END_CFC_
(* the same logic as Structured Text *)
(* result unused: bSetDefault_Global OR HUS2_FA201_FA203._bSetDefault_Plant *)
SERVICEOMKOPPLARE(_bAuto := HUS2_AS01_UPPSTART.START_FA2XX AND bManover, _iMAN := HUS2_FA201_SO1_MAN, _iLM_Delay := HUS2_FA201_SO1_FLM);
bTILL := SERVICEOMKOPPLARE._bStart;
HUS2_FA201_SO1_LM := SERVICEOMKOPPLARE._bLM_DELAYED;
HUS2_FA201_SO1_IA := HUS2_FA201_SO1_MAN = 0;
HUS2_FA201_SO1_IH := HUS2_FA201_SO1_MAN > 0;
HUS2_FA201_SO1_IF := HUS2_FA201_SO1_MAN = 1;
HUS2_FA201_SO1_IT := HUS2_FA201_SO1_MAN = 2;
END_PROGRAM

(* POU SYSTEM/FA201, FA202, FA203/Fläktstyr/HUS2_FA201_FF01, CFC *)
PROGRAM HUS2_FA201_FF01

VAR
	MANHAND: fbManualOverride;





END_VAR
VAR

END_VAR

VAR_INPUT
	_bAuto							:BOOL;(* enable function block *)
END_VAR

VAR_OUTPUT
	_bMANOVER						:BOOL;
	_bLHAND							:BOOL;
END_VAR
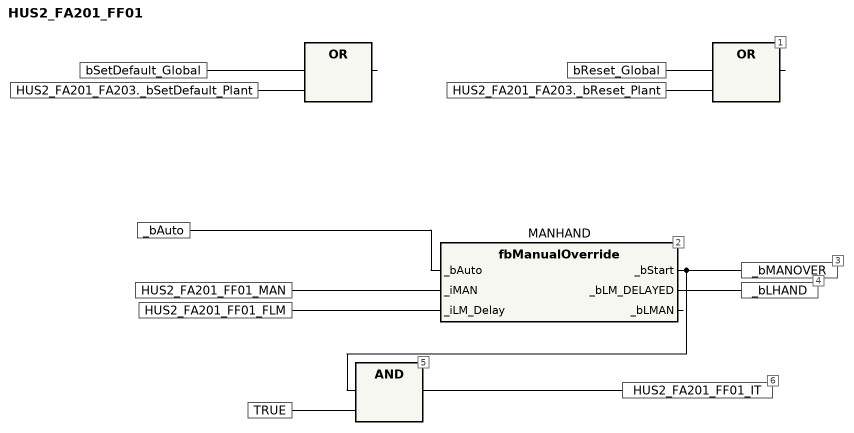
_CFC_ (* Continuous Function Chart, elements in execution order *)
#0 OR(bSetDefault_Global, HUS2_FA201_FA203._bSetDefault_Plant)
#1 OR(bReset_Global, HUS2_FA201_FA203._bReset_Plant)
#2 MANHAND:fbManualOverride(_bAuto: _bAuto, _iMAN: HUS2_FA201_FF01_MAN, _iLM_Delay: HUS2_FA201_FF01_FLM)
#3 _bMANOVER <= #2._bStart
#4 _bLHAND <= #2._bLM_DELAYED
#5 AND(#2._bStart, TRUE)
#6 HUS2_FA201_FF01_IT <= #5
_END_CFC_
(* the same logic as Structured Text *)
(* result unused: bSetDefault_Global OR HUS2_FA201_FA203._bSetDefault_Plant *)
(* result unused: bReset_Global OR HUS2_FA201_FA203._bReset_Plant *)
MANHAND(_bAuto := _bAuto, _iMAN := HUS2_FA201_FF01_MAN, _iLM_Delay := HUS2_FA201_FF01_FLM);
_bMANOVER := MANHAND._bStart;
_bLHAND := MANHAND._bLM_DELAYED;
HUS2_FA201_FF01_IT := MANHAND._bStart AND TRUE;
END_PROGRAM

(* POU SYSTEM/FA201, FA202, FA203/Fläktstyr/HUS2_FA201_FF01_REGLERING, CFC *)
PROGRAM HUS2_FA201_FF01_REGLERING

VAR
	SETRESET: SR;
END_VAR

VAR_INPUT
	bStartFlakt			:BOOL;
	rMV				:REAL;
	rStartForc			:REAL;
	rStoppForc		:REAL;
	rGrundBV			:REAL;
	rForcBV			:REAL;
	bLG				:BOOL;

END_VAR

VAR_OUTPUT
	rSV			:REAL;

END_VAR
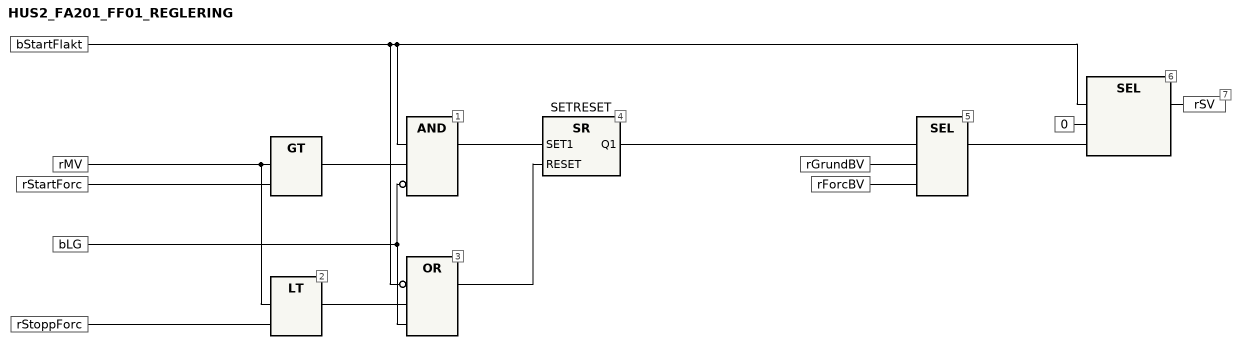
_CFC_ (* Continuous Function Chart, elements in execution order *)
#0 GT(rMV, rStartForc)
#1 AND(bStartFlakt, #0, NOT bLG)
#2 LT(rMV, rStoppForc)
#3 OR(NOT bStartFlakt, #2, bLG)
#4 SETRESET:SR(SET1: #1, RESET: #3)
#5 SEL(#4.Q1, rGrundBV, rForcBV)
#6 SEL(bStartFlakt, 0, #5)
#7 rSV <= #6
_END_CFC_
(* the same logic as Structured Text *)
SETRESET(SET1 := bStartFlakt AND (rMV > rStartForc) AND NOT bLG, RESET := NOT bStartFlakt OR (rMV < rStoppForc) OR bLG);
rSV := SEL(bStartFlakt, 0, SEL(SETRESET.Q1, rGrundBV, rForcBV));
END_PROGRAM

(* POU SYSTEM/FA201, FA202, FA203/Larm/HUS2_FA201_GT51_LARM, FAI *)
PROGRAM HUS2_FA201_GT51_LARM

VAR_OUTPUT
	_bLSumma					: BOOL;	(*Summalarm*)

END_VAR
VAR

	_bSetDefault: 				BOOL;		(*Se default values*)
	fbLarm: fbAvvikelselarm;


	fbHigh: FB_HVACPersistent_Real;
	fbAlarmDelayLH: FB_HVACPersistent_Int;


END_VAR
(* body not read: cfc97 *)
END_PROGRAM

(* POU SYSTEM/FA201, FA202, FA203/HUS2_FA202_SO, CFC *)
PROGRAM HUS2_FA202_SO
VAR_INPUT

	bManover: BOOL;
END_VAR

VAR
	SERVICEOMKOPPLARE: fbManualOverride;

	UPPSTARTSSEKVENSIERING: BOOL;
END_VAR

VAR_OUTPUT
	bTILL:BOOL;

END_VAR
